(******************************************************************************************************************************************)
(****************************				             	Init / Reset Part                                                   *****************************)
(******************************************************************************************************************************************)
IF xSetEnd THEN
	xEnd:=TRUE;
	xInitStep:=FALSE;
	xSetEnd:=FALSE;
	xStop:=FALSE;
	xStartMainPrc:=FALSE;
	xInitMainCtr:=FALSE;
	xStartMainCtr:=FALSE;
	xStart:=FALSE;
	xHardwareError:=FALSE;
	xQuitErr:=FALSE;
	xError:=FALSE;
	iErrorNr:=0;
	xInitError:=FALSE;
	xFreeze:=FALSE;
	xAbord:=FALSE;
	xReset:=FALSE;
END_IF;
END_FUNCTION_BLOCK

(* POU PRG_STATION_LAYER3/FB_STATIONEN/FB_FUNCTION/FB_FctToolFeedReference, ST *)
FUNCTION_BLOCK FB_FctToolFeedReference
VAR_INPUT
	xMicroRodActive: BOOL;		(* choice of the machine MicroWire or MicroRod *)
	xBeckhoffDriveActive: BOOL;	(* choice of the axis Beckhoff or EcoStep *)
	xSafetyCircuitOn:BOOL;			(* state of the safety circuit-->TRUE=Machine current ON, FALSE=Machine current OFF *)
	T_Standard:ST_RETAIN_DATA;							(* Novram data structure for the standard process parameter *)
END_VAR
VAR_IN_OUT
	xStart : BOOL;					(* start the function *)
	xReset : BOOL;				(* reset the function *)
	xStop : BOOL;					(* stop the active function *)
	xQuitErr : BOOL;				(* quit the error caused of the active function *)
	xAbord : BOOL;				(* abord the active function *)
	TAxisToolFeeder:ST_AXIS;		(* data structure for the ToolFeeder axis *)
END_VAR
VAR_OUTPUT
	xEnd : BOOL;					(* state of the function if a active function is ended *)
	xError : BOOL;					(* state of the function if a active function caused an error *)
	iErrorNr : INT;					(* state of the function if a active function caused an error, in this case give the error number *)
END_VAR
VAR
	xHardwareError: BOOL := FALSE;
	xInitError: BOOL := FALSE;
	iStepError: INT := 0;
	xStartMainCtr: BOOL := FALSE;
	xStartMainPrc: BOOL := FALSE;
	xInitMainCtr: BOOL := FALSE;
	iStepPrc: INT := 0;
	xSetEnd: BOOL := FALSE;
	xInitStep: BOOL := FALSE;
	xFreeze: BOOL := FALSE;
	iTmpErrorNr:INT:=0;
	xTmpInit:BOOL;
	iTmp:INT;
END_VAR
(****************************************************************************************************************************************************)
(*******                                This Functionblock define the function for reference the ToolFeeder Axis                                                 ********)
(****************************************************************************************************************************************************)

(******************************************************************************************************************************************)
(****************************				           Reset Function Part                                                 *****************************)
(******************************************************************************************************************************************)
IF xReset AND NOT(xSetEnd) THEN
	xEnd:=FALSE;
	xSetEnd:=TRUE;
END_IF;
(******************************************************************************************************************************************)
(****************************				              Error Controlling Part                                            *****************************)
(******************************************************************************************************************************************)
IF (xHardwareError OR ((TAxisToolFeeder.T_CtrleSingle.xErr) AND xStartMainPrc)) AND NOT(xSetEnd) THEN
	IF NOT(TAxisToolFeeder.T_CtrleSingle.xExecute) THEN
		IF NOT(xInitError) THEN
			iStepError:=100;
			xInitError:=TRUE;
			IF xHardwareError THEN
				iErrorNr:=iTmpErrorNr;
			ELSE
				xHardwareError:=TRUE;	(* Hardware Error *)
			END_IF;
		END_IF;
		CASE iStepError OF
			100:	iStepError:=0;
				xError:=TRUE;
		END_CASE;
		IF xQuitErr THEN
			xSetEnd:=TRUE;
		END_IF;
	END_IF;
END_IF;
(******************************************************************************************************************************************)
(****************************				              Main Controlling Part                                            *****************************)
(******************************************************************************************************************************************)
IF (xStart OR xStartMainCtr) AND NOT(xSetEnd) AND NOT(xHardwareError) THEN
	IF NOT (xInitMainCtr) THEN
		iTmpErrorNr:=0;
		iStepPrc:=100;
		xInitMainCtr:=TRUE;
		xStartMainCtr:=TRUE;
		xStart:=FALSE;
		xEnd:=FALSE;
		xAbord:=FALSE;
		xTmpInit:=FALSE;
	END_IF;
	IF xStop AND NOT(xTmpInit) THEN
		xTmpInit:=TRUE;
		iTmp:=100;
		RETURN;
	END_IF;
	IF xFreeze THEN
		IF xStart AND NOT(xAbord) THEN
			xFreeze:=FALSE;
			xStart:=FALSE;
		END_IF;
		IF xAbord THEN
			xAbord:=FALSE;
			xFreeze:=FALSE;
			xStart:=FALSE;
			xSetEnd:=TRUE;
		END_IF;
		RETURN;
	END_IF;
	IF NOT(xStartMainPrc) AND NOT(xSetEnd) THEN
		xStartMainPrc:=TRUE;
	END_IF;
END_IF;
(******************************************************************************************************************************************)
(****************************				             immediate Stop Part                                              *****************************)
(******************************************************************************************************************************************)
IF xTmpInit AND NOT(xSetEnd) THEN
	IF NOT(xSafetyCircuitOn) THEN
		xTmpInit:=FALSE;
		iTmp:=100;
		xSetEnd:=TRUE;
		RETURN;
	END_IF;
	CASE iTmp OF
		100:	TAxisToolFeeder.T_CtrleSingle.iFunction:=5;
			TAxisToolFeeder.T_CtrleSingle.xExecute:=NOT(TAxisToolFeeder.T_CtrleSingle.xNotMoving);
			iTmp:=200;
			RETURN;
		200:	IF NOT(TAxisToolFeeder.T_CtrleSingle.xExecute) AND TAxisToolFeeder.T_CtrleSingle.xDone THEN
				iTmp:=300;
			END_IF;
			RETURN;
		300:	xTmpInit:=FALSE;
			iTmp:=100;
			xSetEnd:=TRUE;
			RETURN;
	END_CASE;
END_IF;
(******************************************************************************************************************************************)
(****************************				             Main Procedure Part                                             *****************************)
(******************************************************************************************************************************************)
IF xStartMainPrc AND NOT(xSetEnd) AND NOT(xHardwareError) THEN
	CASE iStepPrc OF
		100:	IF NOT(xInitStep) THEN
				xInitStep:=TRUE;
				IF NOT(TAxisToolFeeder.T_CtrleSingle.xDone)THEN
					xHardwareError:=TRUE;
					iTmpErrorNr:=1;
					RETURN;
				END_IF;
				IF NOT(TAxisToolFeeder.T_CtrleSingle.xPower) THEN
					TAxisToolFeeder.T_CtrleSingle.iFunction:=3;
					TAxisToolFeeder.T_CtrleSingle.xExecute:=TRUE;
				END_IF;
			END_IF;
			IF NOT(TAxisToolFeeder.T_CtrleSingle.xExecute) AND TAxisToolFeeder.T_CtrleSingle.xDone THEN
				xStartMainPrc:=FALSE;
				xInitStep:=FALSE;
				iStepPrc:=200;
			END_IF;
		200:	IF NOT(xInitStep) THEN
				xInitStep:=TRUE;
				TAxisToolFeeder.T_CtrleSingle.lrHomingMethode:=5;
				TAxisToolFeeder.T_CtrleSingle.lrHomeSpeedSwitch:=T_Standard.T_TeachINToolFeeder.rRefSpeed;
				TAxisToolFeeder.T_CtrleSingle.lrHomeSpeedZero:=T_Standard.T_TeachINToolFeeder.rRefSpeed / 10.0;
				TAxisToolFeeder.T_CtrleSingle.lrHomeAcceleration:=T_Standard.T_TeachINToolFeeder.rAcceleration;
				TAxisToolFeeder.T_CtrleSingle.iFunction:=9;	(* Reference Axis *)
				TAxisToolFeeder.T_CtrleSingle.xExecute:=TRUE;
			END_IF;
			IF NOT(TAxisToolFeeder.T_CtrleSingle.xExecute) AND TAxisToolFeeder.T_CtrleSingle.xDone THEN
				xStartMainPrc:=FALSE;
				xInitStep:=FALSE;
				iStepPrc:=0;
				xSetEnd:=TRUE;
			END_IF;
	END_CASE;
END_IF;
(******************************************************************************************************************************************)
(****************************				           Parallel Procedure Part                                          *****************************)
(******************************************************************************************************************************************)

(******************************************************************************************************************************************)
(****************************				             	Init / Reset Part                                                   *****************************)
(******************************************************************************************************************************************)
IF xSetEnd THEN
	xEnd:=TRUE;
	xInitStep:=FALSE;
	xSetEnd:=FALSE;
	xStop:=FALSE;
	xStartMainPrc:=FALSE;
	xInitMainCtr:=FALSE;
	xStartMainCtr:=FALSE;
	xStart:=FALSE;
	xHardwareError:=FALSE;
	xQuitErr:=FALSE;
	xError:=FALSE;
	iErrorNr:=0;
	xInitError:=FALSE;
	xFreeze:=FALSE;
	xAbord:=FALSE;
	xReset:=FALSE;
END_IF;
END_FUNCTION_BLOCK

(* POU PRG_STATION_LAYER3/FB_STATIONEN/FB_FUNCTION/FB_FctStopAxisMovement, ST *)
FUNCTION_BLOCK FB_FctStopAxisMovement
VAR_INPUT
	xMicroRodActive: BOOL;		(* choice of the machine MicroWire or MicroRod *)
	xBeckhoffDriveActive: BOOL;	(* choice of the axis Beckhoff or EcoStep *)
	xSafetyCircuitOn:BOOL;			(* state of the safety circuit-->TRUE=Machine current ON, FALSE=Machine current OFF *)
	T_ProcessImageData:ST_RETAIN_DATA_PROCESSIMAGE;	(* Novram data structure for the process parameter *)
	T_Standard:ST_RETAIN_DATA;							(* Novram data structure for the standard process parameter *)
END_VAR
VAR_IN_OUT
	xStart : BOOL;					(* start the function *)
	xReset : BOOL;				(* reset the function *)
	xStop : BOOL;					(* stop the active function *)
	xQuitErr : BOOL;				(* quit the error caused of the active function *)
	xAbord : BOOL;				(* abord the active function *)
	TAxisToolLeft:ST_AXIS;		(* data structure for the ToolLeft axis *)
	TAxisToolCenter:ST_AXIS;		(* data structure for the ToolCenter axis *)
	TAxisToolRight:ST_AXIS;		(* data structure for the ToolRight axis *)
	TAxisToolFeeder:ST_AXIS;		(* data structure for the ToolFeeder axis *)
	TAxisGrindFeeder:ST_AXIS;	(* data structure for the GrindFeeder axis *)
END_VAR
VAR_OUTPUT
	xEnd : BOOL;					(* state of the function if a active function is ended *)
	xError : BOOL;					(* state of the function if a active function caused an error *)
	iErrorNr : INT;					(* state of the function if a active function caused an error, in this case give the error number *)
END_VAR
VAR
	xHardwareError: BOOL := FALSE;
	xInitError: BOOL := FALSE;
	iStepError: INT := 0;
	xStartMainCtr: BOOL := FALSE;
	xStartMainPrc: BOOL := FALSE;
	xInitMainCtr: BOOL := FALSE;
	iStepPrc: INT := 0;
	xSetEnd: BOOL := FALSE;
	xInitStep: BOOL := FALSE;
	xFreeze: BOOL := FALSE;
	iTmpErrorNr:INT:=0;
	xTmpInit:BOOL;
	iTmp:INT;
	xTmp: BOOL;
	xReadFirstTime: BOOL;
	xTmp1: BOOL;
	rToolRotationSpeed: REAL;
	FBToolCalcul:FB_TOOL_CALCUL;
	rToolFeedLength: REAL;
	rToolDiameter: REAL;
	rGrindFeedPlunge: REAL;
	ii: INT;
	iStartSection: INT;
	iEndSection: INT;
	rSpeedGrindFeed: REAL;
	rSpeedToolFeed: REAL;
	rTimeGrindPlunge: REAL;
	FBCalcGearFactor: FB_CALC_GEARFACTOR;
	lrToolFeederActualPosition: LREAL;
	iTmpStartSection: INT;
	FBCalcPlungeGrinding: FB_CALC_PLUNGE_GRINDING;
	xResetFB: BOOL;
	xGrindFeedMaster: BOOL;
	xCheckToolFeedPosition: BOOL;
	lrToolFeederPosition: LREAL;
	lrToolRightPosition: LREAL;
	lrSaveToolFeederPosition: LREAL;
	lrSaveToolRightPosition: LREAL;
	rPlungeCycleGrindFeedGeometry: REAL;
END_VAR
(****************************************************************************************************************************************************)
(***********                               This Functionblock check the movement of all axis and stopp all movement                              ************)
(****************************************************************************************************************************************************)

IF NOT(xReadFirstTime) THEN
	xReadFirstTime:=TRUE;
END_IF;
(******************************************************************************************************************************************)
(****************************				           Reset Function Part                                                 *****************************)
(******************************************************************************************************************************************)
IF xReset AND NOT(xSetEnd) THEN
	xEnd:=FALSE;
	xSetEnd:=TRUE;
END_IF;
(******************************************************************************************************************************************)
(****************************				              Error Controlling Part                                            *****************************)
(******************************************************************************************************************************************)
xTmp:=	TAxisToolLeft.T_CtrleSingle.xErr OR
		(TAxisToolCenter.T_CtrleSingle.xErr AND xMicroRodActive) OR
		TAxisToolRight.T_CtrleSingle.xErr OR
		TAxisToolFeeder.T_CtrleSingle.xErr OR
		TAxisGrindFeeder.T_CtrleSingle.xErr;
xTmp1:=	NOT(TAxisToolLeft.T_CtrleSingle.xExecute) AND
		((NOT(TAxisToolCenter.T_CtrleSingle.xExecute) AND xMicroRodActive) OR NOT(xMicroRodActive)) AND
		 NOT(TAxisToolRight.T_CtrleSingle.xExecute) AND
		((NOT(TAxisToolFeeder.T_CtrleSingle.xExecute) AND NOT(xMicroRodActive)) OR xMicroRodActive) AND
		NOT(TAxisGrindFeeder.T_CtrleSingle.xExecute);
IF (xHardwareError OR (xTmp AND xStartMainPrc)) AND NOT(xSetEnd) THEN
	IF xTmp1 THEN
		IF NOT(xInitError) THEN
			iStepError:=100;
			xInitError:=TRUE;
			IF xHardwareError THEN
				iErrorNr:=iTmpErrorNr;
			ELSE
				xHardwareError:=TRUE;	(* Hardware Error *)
			END_IF;
		END_IF;
		CASE iStepError OF
			100:	iStepError:=0;
				xError:=TRUE;
		END_CASE;
		IF xQuitErr THEN
			xSetEnd:=TRUE;
		END_IF;
	END_IF;
END_IF;
(******************************************************************************************************************************************)
(****************************				              Main Controlling Part                                            *****************************)
(******************************************************************************************************************************************)
IF (xStart OR xStartMainCtr) AND NOT(xSetEnd) AND NOT(xHardwareError) THEN
	IF NOT (xInitMainCtr) THEN
		iTmpErrorNr:=0;
		iStepPrc:=100;
		xInitMainCtr:=TRUE;
		xStartMainCtr:=TRUE;
		xStart:=FALSE;
		xEnd:=FALSE;
		xAbord:=FALSE;
		xTmpInit:=FALSE;
		xCheckToolFeedPosition:=FALSE;
	END_IF;
	IF xStop AND NOT(xTmpInit) THEN
		xTmpInit:=TRUE;
		iTmp:=100;
		RETURN;
	END_IF;
	IF xFreeze THEN
		IF xStart AND NOT(xAbord) THEN
			xFreeze:=FALSE;
			xStart:=FALSE;
		END_IF;
		IF xAbord THEN
			xAbord:=FALSE;
			xFreeze:=FALSE;
			xStart:=FALSE;
			xSetEnd:=TRUE;
		END_IF;
		RETURN;
	END_IF;
	IF NOT(xStartMainPrc) AND NOT(xSetEnd) THEN
		xStartMainPrc:=TRUE;
	END_IF;
END_IF;
(******************************************************************************************************************************************)
(****************************				             immediate Stop Part                                              *****************************)
(******************************************************************************************************************************************)
IF xTmpInit AND NOT(xSetEnd) THEN
	IF NOT(xSafetyCircuitOn) THEN
		xTmpInit:=FALSE;
		iTmp:=100;
		xSetEnd:=TRUE;
		RETURN;
	END_IF;
	CASE iTmp OF
		100:	TAxisToolLeft.T_CtrleSingle.iFunction:=5;
			TAxisToolLeft.T_CtrleSingle.xExecute:=NOT(TAxisToolLeft.T_CtrleSingle.xNotMoving);
			IF xMicroRodActive THEN
				TAxisToolCenter.T_CtrleSingle.iFunction:=5;
				TAxisToolCenter.T_CtrleSingle.xExecute:=NOT(TAxisToolCenter.T_CtrleSingle.xNotMoving);
			END_IF;
			TAxisToolRight.T_CtrleSingle.iFunction:=5;
			TAxisToolRight.T_CtrleSingle.xExecute:=NOT(TAxisToolRight.T_CtrleSingle.xNotMoving);
			TAxisToolFeeder.T_CtrleSingle.iFunction:=5;
			TAxisToolFeeder.T_CtrleSingle.xExecute:=NOT(TAxisToolFeeder.T_CtrleSingle.xNotMoving);
			TAxisGrindFeeder.T_CtrleSingle.iFunction:=5;
			TAxisGrindFeeder.T_CtrleSingle.xExecute:=NOT(TAxisGrindFeeder.T_CtrleSingle.xNotMoving);
			iTmp:=200;
			RETURN;
		200:	xTmp:=	NOT(TAxisToolLeft.T_CtrleSingle.xExecute) AND TAxisToolLeft.T_CtrleSingle.xDone AND
					((NOT(TAxisToolCenter.T_CtrleSingle.xExecute) AND TAxisToolCenter.T_CtrleSingle.xDone AND xMicroRodActive) OR NOT(xMicroRodActive)) AND
					NOT(TAxisToolRight.T_CtrleSingle.xExecute) AND TAxisToolRight.T_CtrleSingle.xDone AND
					NOT(TAxisToolFeeder.T_CtrleSingle.xExecute) AND TAxisToolFeeder.T_CtrleSingle.xDone AND
					NOT(TAxisGrindFeeder.T_CtrleSingle.xExecute) AND TAxisGrindFeeder.T_CtrleSingle.xDone;
			IF xTmp THEN
				iTmp:=300;
			END_IF;
			RETURN;
		300:	IF xMicroRodActive THEN
				IF TAxisToolCenter.T_CtrleSingle.xSlave THEN
					TAxisToolCenter.T_CtrleSingle.iFunction:=25;
					TAxisToolCenter.T_CtrleSingle.xExecute:=TRUE;
				END_IF;
			END_IF;
			IF TAxisToolRight.T_CtrleSingle.xSlave THEN
				TAxisToolRight.T_CtrleSingle.iFunction:=25;
				TAxisToolRight.T_CtrleSingle.xExecute:=TRUE;
			END_IF;
			IF TAxisToolFeeder.T_CtrleSingle.xSlave THEN
				TAxisToolFeeder.T_CtrleSingle.iFunction:=25;
				TAxisToolFeeder.T_CtrleSingle.xExecute:=TRUE;
			END_IF;
			IF TAxisGrindFeeder.T_CtrleSingle.xSlave THEN
				TAxisGrindFeeder.T_CtrleSingle.iFunction:=25;
				TAxisGrindFeeder.T_CtrleSingle.xExecute:=TRUE;
			END_IF;
			iTmp:=400;
			RETURN;
		400:	xTmp:=	((NOT(TAxisToolCenter.T_CtrleSingle.xExecute) AND TAxisToolCenter.T_CtrleSingle.xDone AND xMicroRodActive) OR NOT(xMicroRodActive)) AND
					NOT(TAxisToolRight.T_CtrleSingle.xExecute) AND TAxisToolRight.T_CtrleSingle.xDone AND
					NOT(TAxisToolFeeder.T_CtrleSingle.xExecute) AND TAxisToolFeeder.T_CtrleSingle.xDone AND
					NOT(TAxisGrindFeeder.T_CtrleSingle.xExecute) AND TAxisGrindFeeder.T_CtrleSingle.xDone;
			IF xTmp THEN
				iTmp:=500;
			END_IF;
			RETURN;
		500:	xTmpInit:=FALSE;
			iTmp:=100;
			xSetEnd:=TRUE;
			RETURN;
	END_CASE;
END_IF;
(******************************************************************************************************************************************)
(****************************				             Main Procedure Part                                             *****************************)
(******************************************************************************************************************************************)
IF xStartMainPrc AND NOT(xSetEnd) AND NOT(xHardwareError) THEN
	CASE iStepPrc OF
		(* Initial Procedure *)
		100:	IF NOT(xInitStep) THEN
				xInitStep:=TRUE;
				TAxisToolLeft.T_CtrleSingle.iFunction:=5;
				TAxisToolLeft.T_CtrleSingle.xExecute:=NOT(TAxisToolLeft.T_CtrleSingle.xNotMoving);
				IF xMicroRodActive THEN
					TAxisToolCenter.T_CtrleSingle.iFunction:=5;
					TAxisToolCenter.T_CtrleSingle.xExecute:=NOT(TAxisToolCenter.T_CtrleSingle.xNotMoving);
				END_IF;
				TAxisToolRight.T_CtrleSingle.iFunction:=5;
				TAxisToolRight.T_CtrleSingle.xExecute:=NOT(TAxisToolRight.T_CtrleSingle.xNotMoving);
				TAxisToolFeeder.T_CtrleSingle.iFunction:=5;
				TAxisToolFeeder.T_CtrleSingle.xExecute:=NOT(TAxisToolFeeder.T_CtrleSingle.xNotMoving);
				TAxisGrindFeeder.T_CtrleSingle.iFunction:=5;
				TAxisGrindFeeder.T_CtrleSingle.xExecute:=NOT(TAxisGrindFeeder.T_CtrleSingle.xNotMoving);
			END_IF;
			xTmp:=	NOT(TAxisToolLeft.T_CtrleSingle.xExecute) AND TAxisToolLeft.T_CtrleSingle.xDone AND
					((NOT(TAxisToolCenter.T_CtrleSingle.xExecute) AND TAxisToolCenter.T_CtrleSingle.xDone AND xMicroRodActive) OR NOT(xMicroRodActive)) AND
					NOT(TAxisToolRight.T_CtrleSingle.xExecute) AND TAxisToolRight.T_CtrleSingle.xDone AND
					NOT(TAxisToolFeeder.T_CtrleSingle.xExecute) AND TAxisToolFeeder.T_CtrleSingle.xDone AND
					NOT(TAxisGrindFeeder.T_CtrleSingle.xExecute) AND TAxisGrindFeeder.T_CtrleSingle.xDone;
			IF xTmp THEN
				xStartMainPrc:=FALSE;
				xInitStep:=FALSE;
				iStepPrc:=200;
			END_IF;
		200:	IF NOT(xInitStep) THEN
				xInitStep:=TRUE;
				IF xMicroRodActive THEN
					IF TAxisToolCenter.T_CtrleSingle.xSlave THEN
						TAxisToolCenter.T_CtrleSingle.iFunction:=25;
						TAxisToolCenter.T_CtrleSingle.xExecute:=TRUE;
					END_IF;
				END_IF;
				IF TAxisToolRight.T_CtrleSingle.xSlave THEN
					TAxisToolRight.T_CtrleSingle.iFunction:=25;
					TAxisToolRight.T_CtrleSingle.xExecute:=TRUE;
				END_IF;
				IF TAxisToolFeeder.T_CtrleSingle.xSlave THEN
					TAxisToolFeeder.T_CtrleSingle.iFunction:=25;
					TAxisToolFeeder.T_CtrleSingle.xExecute:=TRUE;
				END_IF;
				IF TAxisGrindFeeder.T_CtrleSingle.xSlave THEN
					TAxisGrindFeeder.T_CtrleSingle.iFunction:=25;
					TAxisGrindFeeder.T_CtrleSingle.xExecute:=TRUE;
				END_IF;
			END_IF;
			xTmp:=	((NOT(TAxisToolCenter.T_CtrleSingle.xExecute) AND TAxisToolCenter.T_CtrleSingle.xDone AND xMicroRodActive) OR NOT(xMicroRodActive)) AND
					NOT(TAxisToolRight.T_CtrleSingle.xExecute) AND TAxisToolRight.T_CtrleSingle.xDone AND
					NOT(TAxisToolFeeder.T_CtrleSingle.xExecute) AND TAxisToolFeeder.T_CtrleSingle.xDone AND
					NOT(TAxisGrindFeeder.T_CtrleSingle.xExecute) AND TAxisGrindFeeder.T_CtrleSingle.xDone;
			IF xTmp THEN
				(* Procedure is finished *)
				xStartMainPrc:=FALSE;
				xInitStep:=FALSE;
				iStepPrc:=0;
				xSetEnd:=TRUE;
			END_IF;
	END_CASE;
END_IF;
(******************************************************************************************************************************************)
(****************************				           Parallel Procedure Part                                          *****************************)
(******************************************************************************************************************************************)
(******************************************************************************************************************************************)
(****************************				             	Init / Reset Part                                                   *****************************)
(******************************************************************************************************************************************)
IF xSetEnd THEN
	xEnd:=TRUE;
	xInitStep:=FALSE;
	xSetEnd:=FALSE;
	xStop:=FALSE;
	xStartMainPrc:=FALSE;
	xInitMainCtr:=FALSE;
	xStartMainCtr:=FALSE;
	xStart:=FALSE;
	xHardwareError:=FALSE;
	xQuitErr:=FALSE;
	xError:=FALSE;
	iErrorNr:=0;
	xInitError:=FALSE;
	xFreeze:=FALSE;
	xAbord:=FALSE;
	xReset:=FALSE;
	xCheckToolFeedPosition:=FALSE;
END_IF;
END_FUNCTION_BLOCK

(* POU PRG_HARDWARE_LAYER2/PRG_HW_GENERAL, FBD *)
PROGRAM PRG_HW_GENERAL
VAR
	FBHWHdd: FBHW_HDD;
	FBNovRam: FBHW_NOVRAM;
	FBDeviceId:FBHW_DEVICEID;
	FBBoxId:FBHW_BOXID;
	FBProfileFile: FB_PROFILE_FILE;
	FBControlLamp: FB_CONTROLLAMP;
	xDeleteThisVariable:BOOL;
END_VAR
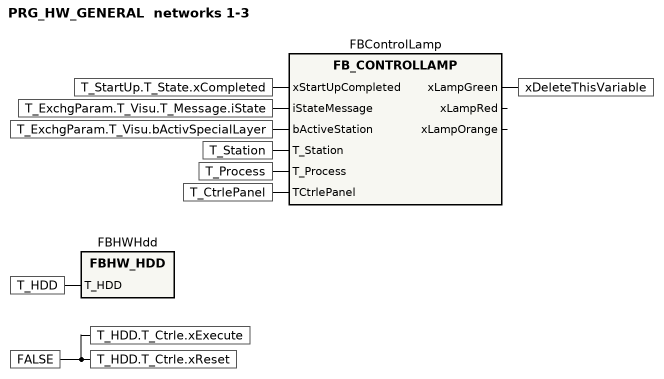
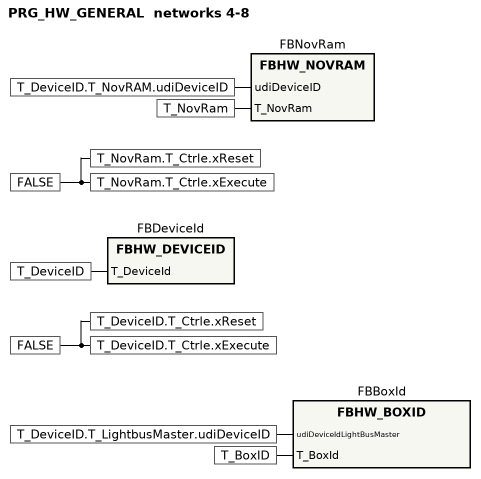
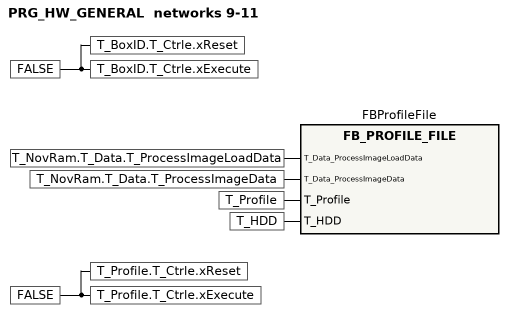
_FBD_ (* Function Block Diagram *)
NETWORK 1
	FBControlLamp:FB_CONTROLLAMP(xStartUpCompleted: T_StartUp.T_State.xCompleted, iStateMessage: T_ExchgParam.T_Visu.T_Message.iState, bActiveStation: T_ExchgParam.T_Visu.bActivSpecialLayer, T_Station: T_Station, T_Process: T_Process, TCtrlePanel: T_CtrlePanel) => xDeleteThisVariable
NETWORK 2
	FBHWHdd:FBHW_HDD(T_HDD: T_HDD)
NETWORK 3
	FALSE => T_HDD.T_Ctrle.xExecute, T_HDD.T_Ctrle.xReset
NETWORK 4
	FBNovRam:FBHW_NOVRAM(udiDeviceID: T_DeviceID.T_NovRAM.udiDeviceID, T_NovRam: T_NovRam)
NETWORK 5
	FALSE => T_NovRam.T_Ctrle.xReset, T_NovRam.T_Ctrle.xExecute
NETWORK 6
	FBDeviceId:FBHW_DEVICEID(T_DeviceId: T_DeviceID)
NETWORK 7
	FALSE => T_DeviceID.T_Ctrle.xReset, T_DeviceID.T_Ctrle.xExecute
NETWORK 8
	FBBoxId:FBHW_BOXID(udiDeviceIdLightBusMaster: T_DeviceID.T_LightbusMaster.udiDeviceID, T_BoxId: T_BoxID)
NETWORK 9
	FALSE => T_BoxID.T_Ctrle.xReset, T_BoxID.T_Ctrle.xExecute
NETWORK 10
	FBProfileFile:FB_PROFILE_FILE(T_Data_ProcessImageLoadData: T_NovRam.T_Data.T_ProcessImageLoadData, T_Data_ProcessImageData: T_NovRam.T_Data.T_ProcessImageData, T_Profile: T_Profile, T_HDD: T_HDD)
NETWORK 11
	FALSE => T_Profile.T_Ctrle.xReset, T_Profile.T_Ctrle.xExecute
_END_FBD_
(* the same logic as Structured Text *)
(* Network 1 *)
FBControlLamp(xStartUpCompleted := T_StartUp.T_State.xCompleted, iStateMessage := T_ExchgParam.T_Visu.T_Message.iState, bActiveStation := T_ExchgParam.T_Visu.bActivSpecialLayer, T_Station := T_Station, T_Process := T_Process, TCtrlePanel := T_CtrlePanel);
xDeleteThisVariable := FBControlLamp.xLampGreen;
(* Network 2 *)
FBHWHdd(T_HDD := T_HDD);
(* Network 3 *)
T_HDD.T_Ctrle.xExecute := FALSE;
T_HDD.T_Ctrle.xReset := FALSE;
(* Network 4 *)
FBNovRam(udiDeviceID := T_DeviceID.T_NovRAM.udiDeviceID, T_NovRam := T_NovRam);
(* Network 5 *)
T_NovRam.T_Ctrle.xReset := FALSE;
T_NovRam.T_Ctrle.xExecute := FALSE;
(* Network 6 *)
FBDeviceId(T_DeviceId := T_DeviceID);
(* Network 7 *)
T_DeviceID.T_Ctrle.xReset := FALSE;
T_DeviceID.T_Ctrle.xExecute := FALSE;
(* Network 8 *)
FBBoxId(udiDeviceIdLightBusMaster := T_DeviceID.T_LightbusMaster.udiDeviceID, T_BoxId := T_BoxID);
(* Network 9 *)
T_BoxID.T_Ctrle.xReset := FALSE;
T_BoxID.T_Ctrle.xExecute := FALSE;
(* Network 10 *)
FBProfileFile(T_Data_ProcessImageLoadData := T_NovRam.T_Data.T_ProcessImageLoadData, T_Data_ProcessImageData := T_NovRam.T_Data.T_ProcessImageData, T_Profile := T_Profile, T_HDD := T_HDD);
(* Network 11 *)
T_Profile.T_Ctrle.xReset := FALSE;
T_Profile.T_Ctrle.xExecute := FALSE;
END_PROGRAM

(* POU FB_HARDWARE/FBHW_HDD, ST *)
FUNCTION_BLOCK FBHW_HDD
VAR_INPUT
END_VAR
VAR_OUTPUT
END_VAR
VAR_IN_OUT
	T_HDD:ST_HDD;
END_VAR
VAR
(* variable *)
	xConfirmResetFB: BOOL;
	i:INT;
	dwOpenFileMod:DWORD;
	udiHdleFile:UINT;
	xFileOpen: BOOL;
	xFileClose:BOOL;
	xFileRead:BOOL;
	xFileAppendWrite:BOOL;
	xFileCreate:BOOL;
	xFileBiggerAsMaxLine:BOOL;
	xFileDelete: BOOL;
	xRenameFile:BOOL;

(* function bloc *)
	fbFileOpen:FB_FileOpen;
	fbFileWrite:FB_FileWrite;

	fbFileClose:FB_FileClose;
	fbFileGets:FB_FileGets;
	fbFilePuts:FB_FilePuts;

	fbFileDelete:FB_FileDelete;
	fbRenameFile:FB_FileRename;
(* Trigger *)
	RisingEdgeExecute:R_TRIG;
	RisingEdgeReset:R_TRIG;
END_VAR
(****************************************************************************************************************************************************)
(***********                                                  This Functionblock is for manage the file handling                                                             ************)
(****************************************************************************************************************************************************)
(* waiting for reset *)
	RisingEdgeReset(CLK:=T_HDD.T_Ctrle.xReset);
	IF RisingEdgeReset.Q THEN
	(* init. function bloc *)
		fbFileOpen(bExecute:=FALSE);
		fbFileClose(bExecute:=FALSE);
		fbFileWrite(bExecute:=FALSE);
		fbFileGets(bExecute:=FALSE);
		fbFilePuts(bExecute:=FALSE);
		fbFileDelete(bExecute:=FALSE);
		fbRenameFile(bExecute:=FALSE);
	(* init. variable *)
		dwOpenFileMod:=0;
		udiHdleFile:=0;
		xFileOpen:=FALSE;
		xFileClose:=FALSE;
		xFileRead:=FALSE;
		xFileAppendWrite:=FALSE;
		xFileCreate:=FALSE;
		xFileBiggerAsMaxLine:=FALSE;
		xFileDelete:=FALSE;
		xRenameFile:=FALSE;
	(* init. structure *)
		T_HDD.T_Ctrle.xDone:=FALSE;
		T_HDD.T_Ctrle.xErr:=FALSE;
		T_HDD.T_Ctrle.udiErrorID:=0;
		T_HDD.T_Ctrle.iFunction:=0;
		T_HDD.T_File.sPathAndFileName:='';
		T_HDD.T_File.sOldPathAndFileName:='';
		T_HDD.T_Ctrle.tTimeOut:=T#2s;
		T_HDD.T_Ctrle.xLocked:=FALSE;
		(* set flag done *)
		xConfirmResetFB:=TRUE;
		(* exit function *)
		RETURN;
	ELSE
		IF xConfirmResetFB THEN
		(* confirm reset FB *)
			T_HDD.T_Ctrle.xDone:=TRUE;
			T_HDD.T_Ctrle.xErr:=FALSE;
			T_HDD.T_Ctrle.udiErrorID:=0;
			T_HDD.T_Ctrle.xLocked:=FALSE;
			(* init. variable *)
			xConfirmResetFB:=FALSE;
		END_IF
	END_IF

(* waiting for execute *)
	RisingEdgeExecute(CLK:=T_HDD.T_Ctrle.xExecute);
	IF RisingEdgeExecute.Q THEN
		CASE T_HDD.T_Ctrle.iFunction OF
		(* Read file *)
		1:	(* activ file open *)
			xFileOpen:=TRUE;
			dwOpenFileMod:=FOPEN_MODEREAD OR FOPEN_MODEPLUS OR FOPEN_MODETEXT;
		(* Write file *)
		2:	(* activ file open *)
			xFileOpen:=TRUE;
			dwOpenFileMod:=FOPEN_MODEWRITE OR FOPEN_MODEPLUS OR FOPEN_MODETEXT;
		(* overwrite file *)
		3:	(* activ file open *)
			xFileOpen:=TRUE;
			dwOpenFileMod:=FOPEN_MODEAPPEND OR FOPEN_MODEPLUS OR FOPEN_MODETEXT;
		(* file exists *)
		4:	(* activ file open *)
			xFileOpen:=TRUE;
			dwOpenFileMod:=FOPEN_MODEREAD OR FOPEN_MODEPLUS OR FOPEN_MODETEXT;
		(* delete file *)
		5:	xFileDelete:=TRUE;
		(* rename file *)
		6:	xRenameFile:=TRUE;
		ELSE
		(* function not implemented *)
			 T_HDD.T_Ctrle.xDone:=FALSE;
			 T_HDD.T_Ctrle.xErr:=TRUE;
			 T_HDD.T_Ctrle.udiErrorID:=16#F000;
			 T_HDD.T_Ctrle.xLocked:=FALSE;
			 (* exit FB *)
			 RETURN;
		END_CASE
		(* Init. variable *)
		T_HDD.T_Ctrle.xDone:=FALSE;
		T_HDD.T_Ctrle.xErr:=FALSE;
		T_HDD.T_Ctrle.udiErrorID:=16#0;
		xFileBiggerAsMaxLine:=FALSE;
		(* init. variable*)
		i:=1;
		RETURN;
	END_IF

(* Open file *)
	IF xFileOpen THEN
		fbFileOpen(	sNetId:=T_HDD.T_Config.sNetId,
					sPathName:=T_HDD.T_File.sPathAndFileName,
					nMode:=dwOpenFileMod,
					bExecute:=TRUE,
					tTimeout:=T#2s);
		IF NOT(fbFileOpen.bBusy) OR fbFileOpen.bError THEN
			IF NOT(fbFileOpen.bError) THEN
				CASE T_HDD.T_Ctrle.iFunction OF
				1:	xFileRead:=TRUE;
				2:	xFileCreate:=TRUE;
				3: 	xFileAppendWrite:=TRUE;
				4:	xFileClose:=TRUE;
				END_CASE
				(* Handle file *)
				udiHdleFile:=fbFileOpen.hFile;
			ELSE
				udiHdleFile:=0;
				 T_HDD.T_Ctrle.xDone:= FALSE;
				 T_HDD.T_Ctrle.xErr:=fbFileOpen.bError;
				 T_HDD.T_Ctrle.udiErrorID:=fbFileOpen.nErrId;
				 T_HDD.T_Ctrle.xLocked:=FALSE;
			END_IF
			(* set flag xfileopen off *)
			xFileOpen:=FALSE;
		END_IF
	ELSE fbFileOpen(bExecute:=FALSE); END_IF

(* Read file *)
	IF xFileRead THEN
		fbFileGets(	sNetId:=T_HDD.T_Config.sNetId,
					hFile:=udiHdleFile,
					bExecute:=TRUE,
					tTimeOut:=T_HDD.T_Ctrle.tTimeOut);
		IF NOT(fbFileGets.bBusy) OR fbFileGets.bError THEN
			T_HDD.T_Data.sData[i]:=fbFileGets.sLine;
			(* check eof or error *)
			IF fbFileGets.bEOF OR fbFileGets.bError OR i = csiMaxFileLine THEN
				 (* set flag xFileRead off *)
				 xFileRead:=FALSE;
				 (* activ closing file *)
				 xFileClose:=TRUE;
				 (* activ variable file bigger as structure *)
				 IF i = csiMaxFileLine THEN xFileBiggerAsMaxLine:=TRUE; END_IF
			ELSE
			(* read next line *)
				fbFileGets(bExecute:=FALSE);
				i:=i+1;
			END_IF
		END_IF
	ELSE fbFileGets(bExecute:=FALSE); END_IF

(* Write at the end of file or create file *)
	IF xFileAppendWrite OR xFileCreate THEN
		fbFilePuts(	sNetId:=T_HDD.T_Config.sNetId,
					hFile:=udiHdleFile,
					sLine:=CONCAT(T_HDD.T_Data.sData[i],'$L'),
					bExecute:=TRUE,
					tTimeOut:=T_HDD.T_Ctrle.tTimeOut);
		IF NOT(fbFilePuts.bBusy) OR fbFilePuts.bError THEN
			IF T_HDD.T_Data.sData[i+1] = '' THEN
				 (* set flag xFileCreate or xFileAppendWrite off *)
				xFileAppendWrite:=FALSE;
				xFileCreate:=FALSE;
				 (* activ closing file *)
				 xFileClose:=TRUE;
			ELSE
			(* Init. FB *)
				 fbFilePuts(bExecute:=FALSE);
				 (* next line *)
				i:=i+1;
			END_IF
		END_IF
	ELSE IF NOT(xFileAppendWrite) AND NOT(xFileCreate) THEN fbFilePuts(bExecute:=FALSE); END_IF
	END_IF

(* Close file *)
	IF xFileClose THEN
		fbFileClose(	sNetId:=T_HDD.T_Config.sNetId,
					hFile:=udiHdleFile,
					bExecute:=TRUE,
					tTimeout:=T#2s);
		IF NOT(fbFileClose.bBusy) OR fbFileClose.bError THEN
			 T_HDD.T_Ctrle.xDone:= NOT(fbFileClose.bBusy);
			 T_HDD.T_Ctrle.xErr:=fbFileClose.bError;
			 T_HDD.T_Ctrle.udiErrorID:=fbFileClose.nErrId;
			T_HDD.T_Ctrle.xLocked:=FALSE;
			 udiHdleFile:=0;
			(* check if file bigger as maximum reading line *)
			IF xFileBiggerAsMaxLine THEN
				T_HDD.T_Ctrle.xErr:=TRUE;
				T_HDD.T_Ctrle.udiErrorID:=16#F501;
			END_IF
			 (* set flag xFileClose off *)
			 xFileClose:=FALSE;
		END_IF
	ELSE fbFileClose(bExecute:=FALSE); END_IF

(* Delete file *)
	IF xFileDelete THEN
		fbFileDelete(	sNetId:=T_HDD.T_Config.sNetId,
					sPathName:=T_HDD.T_File.sPathAndFileName,
					bExecute:=TRUE,
					tTimeout:=T#2s);
		IF NOT(fbFileDelete.bBusy) OR fbFileDelete.bError THEN
			 T_HDD.T_Ctrle.xDone:= NOT(fbFileDelete.bBusy);
			 T_HDD.T_Ctrle.xErr:=fbFileDelete.bError;
			 T_HDD.T_Ctrle.udiErrorID:=fbFileDelete.nErrId;
			T_HDD.T_Ctrle.xLocked:=FALSE;
			 (* set flag xFileDelete off *)
			 xFileDelete:=FALSE;
		END_IF
	ELSE fbFileDelete(bExecute:=FALSE); END_IF

(* rename file *)
	IF xRenameFile THEN
		fbRenameFile(	sNetId:=T_HDD.T_Config.sNetId,
						sOldName:=T_HDD.T_File.sOldPathAndFileName,
						sNewName:=T_HDD.T_File.sPathAndFileName,
						ePath:=PATH_GENERIC,
						bExecute:=TRUE,
						tTimeout:=T#2s);
		IF NOT(fbRenameFile.bBusy) OR fbRenameFile.bError THEN
			 T_HDD.T_Ctrle.xDone:= NOT(fbRenameFile.bBusy);
			 T_HDD.T_Ctrle.xErr:=fbRenameFile.bError;
			 T_HDD.T_Ctrle.udiErrorID:=fbRenameFile.nErrId;
			T_HDD.T_Ctrle.xLocked:=FALSE;
			 (* set flag xFileDelete off *)
			 xRenameFile:=FALSE;
		END_IF
	ELSE fbRenameFile(bExecute:=FALSE); END_IF
END_FUNCTION_BLOCK

(* POU FB_HARDWARE/FBHW_NOVRAM, ST *)
FUNCTION_BLOCK FBHW_NOVRAM
VAR_INPUT
	udiDeviceID:UDINT;
END_VAR
VAR_IN_OUT
	T_NovRam:ST_NOVRAM;
END_VAR
VAR_OUTPUT
END_VAR
VAR
(* function bloc *)
	fbNovRamReadWrite:FB_NovRamReadWrite;
(* trigger *)
	RisingEdgeResetFB:R_TRIG;
	RisingEdgeExecute:R_TRIG;
(* variable *)
	xRead:BOOL:=FALSE;
	xWrite:BOOL:=FALSE;
	xConfirmResetFB: BOOL;
	xDummy1: BOOL;
	xDummy2: BOOL;
END_VAR
(****************************************************************************************************************************************************)
(***********                                            This Functionblock is for manage the NovRAM handling                                                      ************)
(****************************************************************************************************************************************************)
(* reset *)
	RisingEdgeResetFB(CLK:=T_NovRam.T_Ctrle.xReset);
	IF RisingEdgeResetFB.Q THEN
	(* init. variable *)
		xRead:=FALSE;
		xWrite:=FALSE;
	(* activ confirmation reset *)
		xConfirmResetFB:=TRUE;
	(* Exit FB *)
		RETURN;
	ELSE
		IF xConfirmResetFB THEN
		(* confirm reset FB *)
			T_NovRam.T_Ctrle.xFirstRead:=FALSE;
			T_NovRam.T_Ctrle.xDone:=TRUE;
			T_NovRam.T_Ctrle.xErr:=FALSE;
			T_NovRam.T_Ctrle.udiErrorID:=16#0;
		(* reset variable *)
			xConfirmResetFB:=FALSE;
		END_IF
	END_IF

(* execute *)
	RisingEdgeExecute(CLK:=T_NovRam.T_Ctrle.xExecute);
	IF RisingEdgeExecute.Q THEN
		(* init. capacity and pointer *)
		T_NovRam.T_Ctrle.udipSrcAddr:=ADR(T_NovRam.T_Data);
		T_NovRam.T_Ctrle.udiSrcLen:=SIZEOF(T_NovRam.T_Data);
		T_NovRam.T_Ctrle.udipDestAddr:=ADR(T_NovRam.T_Data);
		T_NovRam.T_Ctrle.udiDestLen:=SIZEOF(T_NovRam.T_Data);
		CASE T_NovRam.T_Ctrle.iFunction OF
		(* Read *)
		1:	xRead:=TRUE;
		(* Write *)
		2:	xWrite:=TRUE;
		ELSE
		(* function not implemented *)
			T_NovRam.T_Ctrle.xDone:=FALSE;
			T_NovRam.T_Ctrle.xErr:=TRUE;
			T_NovRam.T_Ctrle.udiErrorID:=16#F000;
			(* Exit FB *)
			RETURN;
		END_CASE
		(* Init. variable *)
		T_NovRam.T_Ctrle.xDone:=FALSE;
		T_NovRam.T_Ctrle.xErr:=FALSE;
		T_NovRam.T_Ctrle.udiErrorID:=0;
	(* Exit FB *)
		RETURN;
	END_IF

(* wait for read/write *)
	IF xRead OR xWrite THEN
		IF xWrite THEN
			xDummy1:=TRUE;
			xDummy2:=FALSE;
		END_IF;
		IF xRead THEN
			xDummy2:=TRUE;
			xDummy1:=FALSE;
		END_IF;
		fbNovRamReadWrite(	nDevId:=udiDeviceID,
							bRead:=xRead,
							bWrite:=xWrite,
							cbSrcLen:=T_NovRam.T_Ctrle.udiSrcLen,
							cbDestLen:=T_NovRam.T_Ctrle.udiDestLen,
							pSrcAddr:=T_NovRam.T_Ctrle.udipSrcAddr,
							pDestAddr:=T_NovRam.T_Ctrle.udipDestAddr,
							tTimeOut:=T_NovRam.T_Ctrle.tTimeOut);
		IF NOT(fbNovRamReadWrite.bBusy) OR fbNovRamReadWrite.bError THEN
			IF fbNovRamReadWrite.bError THEN
			(* set error *)
				T_NovRam.T_Ctrle.xDone:=FALSE;
				T_NovRam.T_Ctrle.xErr:=TRUE;
				T_NovRam.T_Ctrle.udiErrorID:=fbNovRamReadWrite.nErrId;
			ELSE
			(* confirm execution *)
				IF xRead THEN
					IF NOT(T_NovRam.T_Ctrle.xBlockReadFirstTime) THEN
						T_NovRam.T_Ctrle.xFirstRead:=TRUE;
					ELSE
						T_NovRam.T_Ctrle.xFirstRead:=FALSE;
					END_IF;
					T_NovRam.T_Ctrle.xBlockReadFirstTime:=FALSE;
				END_IF
				T_NovRam.T_Ctrle.xDone:=TRUE;
				T_NovRam.T_Ctrle.xErr:=FALSE;
				T_NovRam.T_Ctrle.udiErrorID:=0;
			END_IF
			(* reset variable *)
			xRead:=FALSE;
			xWrite:=FALSE;
		END_IF
	ELSE
		fbNovRamReadWrite(	nDevId:=udiDeviceID,
							bRead:=FALSE,
							bWrite:=FALSE);
	END_IF
END_FUNCTION_BLOCK

(* POU FB_HARDWARE/FBHW_DEVICEID, ST *)
FUNCTION_BLOCK FBHW_DEVICEID
VAR_INPUT
END_VAR
VAR_IN_OUT
	T_DeviceId:ST_DEVICEID;
END_VAR
VAR_OUTPUT
END_VAR
VAR
(* pointer of Device ID *)
	ptrDeviceId: POINTER TO ST_DEVICEID;
(* function bloc *)
	FBGeviceInfoByName:IOF_GetDeviceInfoByName;
(* trigger *)
	RisingEdgeResetFB:R_TRIG;
	RisingEdgeExecute:R_TRIG;
	FallingEdgeBusy:F_TRIG;
(* variable *)
	xGetDeviceId:BOOL:=FALSE;
	xConfirmResetFB:BOOL:=FALSE;
	iPtrDeviceName:INT:=0;
	T_DeviceId_AdrTmp:ARRAY[1..10] OF ST_DEVICEID_DATA_ADR;
	xInitReadStructure: BOOL;
	xCopyReadyStructure:BOOL;
END_VAR
(****************************************************************************************************************************************************)
(***********                                                This Functionblock is for init the Beckhoff component                                                          ************)
(****************************************************************************************************************************************************)
(* reset *)
	RisingEdgeResetFB(CLK:=T_DeviceId.T_Ctrle.xReset);
	IF RisingEdgeResetFB.Q THEN
	(* init ptr*)
		ptrDeviceId:=ADR(T_DeviceId);
	(* init. variable *)
		xGetDeviceId:=FALSE;
		iPtrDeviceName:=1;
	(* Init. variable *)
		ptrDeviceId^.T_Ctrle.xDone:=FALSE;
		ptrDeviceId^.T_Ctrle.xErr:=FALSE;
		ptrDeviceId^.T_Ctrle.udiErrorID:=0;
	(* activ confirm reset *)
		xConfirmResetFB:=TRUE;
	(* Exit FB *)
		RETURN;
	ELSE
		IF xConfirmResetFB THEN
		(* confirm reset FB *)
			ptrDeviceId^.T_Ctrle.xDone:=TRUE;
			ptrDeviceId^.T_Ctrle.xErr:=FALSE;
			ptrDeviceId^.T_Ctrle.udiErrorID:=0;
		(* reset variable *)
			xConfirmResetFB:=FALSE;
		END_IF
	END_IF

(* execute *)
	RisingEdgeExecute(CLK:=T_DeviceId.T_Ctrle.xExecute);
	IF RisingEdgeExecute.Q THEN
	(* init ptr*)
		ptrDeviceId:=ADR(T_DeviceId);
		ptrDeviceId^.T_Ctrle.xDone:=FALSE;
		ptrDeviceId^.T_Ctrle.xErr:=FALSE;
		ptrDeviceId^.T_Ctrle.udiErrorID:=0;
	(* activ get device Id *)
		xInitReadStructure:=TRUE;
	(* Exit FB *)
		RETURN;
	END_IF

(* init. read structure *)
	IF xInitReadStructure THEN
	(* PLC name *)
		T_DeviceId_AdrTmp[1]:=T_DeviceId.T_CX1020;
		(* feldbus name *)
		T_DeviceId_AdrTmp[2]:=T_DeviceId.T_CANOpenMaster;
		T_DeviceId_AdrTmp[4]:=T_DeviceId.T_LightbusMaster;
		(* NovRAM name *)
		T_DeviceId_AdrTmp[3]:=T_DeviceId.T_NovRAM;
		(* end *)
		T_DeviceId_AdrTmp[5].sDeviceName:='';
		(*reset variable*)
		xInitReadStructure:=FALSE;
		iPtrDeviceName:=1;
		(* start device id reading *)
		xGetDeviceId:=TRUE;
	(* Exit FB *)
		RETURN;
	END_IF

(* get device Id *)
	IF xGetDeviceId THEN
		FallingEdgeBusy(CLK:=FBGeviceInfoByName.BUSY);
		IF FallingEdgeBusy.Q THEN
		(* save device id *)
			T_DeviceId_AdrTmp[iPtrDeviceName].udiDeviceID:=FBGeviceInfoByName.DEVICEID;
			T_DeviceId_AdrTmp[iPtrDeviceName].sAmsNetId:=FBGeviceInfoByName.DEVICENETID;
			(* next device *)
			iPtrDeviceName:=iPtrDeviceName+1;
		END_IF
		IF NOT(FBGeviceInfoByName.BUSY) AND T_DeviceId_AdrTmp[iPtrDeviceName].sDeviceName <> '' THEN
			FBGeviceInfoByName(	NETID:='',
								DEVICENAME:=T_DeviceId_AdrTmp[iPtrDeviceName].sDeviceName,
								START:=TRUE,
								TMOUT:=T#2s);
		ELSE
			FBGeviceInfoByName(START:=FALSE);
		END_IF
		IF NOT(FBGeviceInfoByName.BUSY) AND NOT(FBGeviceInfoByName.ERR) AND T_DeviceId_AdrTmp[iPtrDeviceName].sDeviceName = '' THEN
			(* init. variable *)
			xGetDeviceId:=FALSE;
			(* set copy value *)
			xCopyReadyStructure:=TRUE;
		END_IF
		IF FBGeviceInfoByName.ERR THEN
		(* acitve error *)
			IF NOT(T_DeviceId_AdrTmp[iPtrDeviceName].xDeviceOption) THEN
				IF (iPtrDeviceName <> 5) THEN
					ptrDeviceId^.T_Ctrle.xDone:=FALSE;
					ptrDeviceId^.T_Ctrle.xErr:=TRUE;
					ptrDeviceId^.T_Ctrle.udiErrorID:=FBGeviceInfoByName.ERRID;
					(* init. variable *)
					xGetDeviceId:=FALSE;
				ELSE
					(* init. variable *)
					xGetDeviceId:=FALSE;
					(* set copy value *)
					xCopyReadyStructure:=TRUE;
				END_IF;
			END_IF
		END_IF
	ELSE
		FBGeviceInfoByName(START:=FALSE);
	END_IF

(* copy read value *)
	IF xCopyReadyStructure THEN
	(* copy value *)
		(* PLC name *)
		T_DeviceId.T_CX1020:=T_DeviceId_AdrTmp[1];
		(* feldbus name *)
		T_DeviceId.T_CANOpenMaster:=T_DeviceId_AdrTmp[2];
		T_DeviceId.T_LightbusMaster:=T_DeviceId_AdrTmp[4];
		(* NovRAM name *)
		T_DeviceId.T_NovRAM:=T_DeviceId_AdrTmp[3];
		(* confirm device list id *)
		ptrDeviceId^.T_Ctrle.xDone:=TRUE;
		ptrDeviceId^.T_Ctrle.xErr:=FALSE;
		ptrDeviceId^.T_Ctrle.udiErrorID:=0;
		(* reset variable *)
		xCopyReadyStructure:=FALSE;
	END_IF
END_FUNCTION_BLOCK

(* POU FB_HARDWARE/FBHW_BOXID, ST *)
FUNCTION_BLOCK FBHW_BOXID
VAR_INPUT
	udiDeviceIdLightBusMaster:UDINT;
END_VAR
VAR_IN_OUT
	T_BoxId:ST_BOXID;
END_VAR
VAR_OUTPUT
END_VAR
VAR
(* pointer of Box ID *)
	ptrBoxId: POINTER TO ST_BOXID;
(* function bloc *)
	fbGetBoxAddrByName:IOF_GetBoxAddrByName;
	fbGetBoxNetId:IOF_GetBoxNetId;
(* trigger *)
	RisingEdgeResetFB:R_TRIG;
	RisingEdgeExecute:R_TRIG;
(* variable *)
	xGetBoxId:BOOL:=FALSE;
	xConfirmResetFB:BOOL:=FALSE;
	iPtrBoxName:INT:=0;
	iPtrBoxNameEnd:INT:=0;
	T_BoxId_AdrTmp:ARRAY[1..20] OF ST_BOXID_DATA_ADR;
	xInitReadStructure: BOOL;
	xCopyReadyStructure:BOOL;
	xGetBoxAddress: BOOL;
END_VAR
(****************************************************************************************************************************************************)
(***********                     This Functionblock is needed for read the BoxID information of the Beckhoff components               ************)
(****************************************************************************************************************************************************)
(* reset *)
	RisingEdgeResetFB(CLK:=T_BoxId.T_Ctrle.xReset);
	IF RisingEdgeResetFB.Q THEN
	(* init ptr*)
		ptrBoxId:=ADR(T_BoxId);
	(* init. variable *)
		xGetBoxId:=FALSE;
		iPtrBoxName:=1;
	(* Init. variable *)
		ptrBoxId^.T_Ctrle.xDone:=FALSE;
		ptrBoxId^.T_Ctrle.xErr:=FALSE;
		ptrBoxId^.T_Ctrle.udiErrorID:=0;
	(* activ confirm reset *)
		xConfirmResetFB:=TRUE;
	(* Exit FB *)
		RETURN;
	ELSE
		IF xConfirmResetFB THEN
		(* confirm reset FB *)
			ptrBoxId^.T_Ctrle.xDone:=TRUE;
			ptrBoxId^.T_Ctrle.xErr:=FALSE;
			ptrBoxId^.T_Ctrle.udiErrorID:=0;
		(* reset variable *)
			xConfirmResetFB:=FALSE;
		END_IF
	END_IF

(* execute *)
	RisingEdgeExecute(CLK:=T_BoxId.T_Ctrle.xExecute);
	IF RisingEdgeExecute.Q THEN
	(* init ptr*)
		ptrBoxId:=ADR(T_BoxId);
	(* activ get device Id *)
		xInitReadStructure:=TRUE;
	(* init. state flag *)
		ptrBoxId^.T_Ctrle.xDone:=FALSE;
		ptrBoxId^.T_Ctrle.xErr:=FALSE;
		ptrBoxId^.T_Ctrle.udiErrorID:=0;
	(* Exit FB *)
		RETURN;
	END_IF

(* init. read structure *)
	IF xInitReadStructure THEN
	(* PLC name, servo  *)
		iPtrBoxName:=1;
		T_BoxId_AdrTmp[1]:=T_BoxId.T_Servo_ToolLeft;
		T_BoxId_AdrTmp[2]:=T_BoxId.T_Servo_ToolCenter;
		T_BoxId_AdrTmp[3]:=T_BoxId.T_Servo_ToolRight;
		T_BoxId_AdrTmp[4]:=T_BoxId.T_Servo_ToolFeeder;
		T_BoxId_AdrTmp[5]:=T_BoxId.T_Servo_GrindFeeder;
		iPtrBoxNameEnd:=5;
		(* end *)
		T_BoxId_AdrTmp[6].sDeviceName:='';
		(*reset variable*)
		xInitReadStructure:=FALSE;
		(* start device id reading *)
		xGetBoxAddress:=TRUE;
	(* Exit FB *)
		RETURN;
	END_IF

(* get box address *)
	IF xGetBoxAddress THEN
		fbGetBoxAddrByName(	NETID:='',
								DEVICEID:=udiDeviceIdLightBusMaster,
								BOXNAME:=T_BoxId_AdrTmp[iPtrBoxName].sBoxName,
								START:=TRUE,
								TMOUT:=T#2s);
		IF NOT(fbGetBoxAddrByName.BUSY) OR fbGetBoxAddrByName.ERR THEN
			IF fbGetBoxAddrByName.ERR THEN
				IF T_BoxId_AdrTmp[iPtrBoxName].xDeviceOption THEN
				(* Init. FB *)
					fbGetBoxAddrByName(START:=FALSE);
					IF iPtrBoxName <> iPtrBoxNameEnd THEN
					(* next box *)
						iPtrBoxName:=iPtrBoxName+1;
						IF (T_BoxId.T_Ctrle.iMachineType = 1) AND (iPtrBoxName = 2) THEN
							iPtrBoxName:=3;
						END_IF;
						(* exit FB *)
						RETURN;
					(* activ copy value *)
					ELSE xCopyReadyStructure:=TRUE;END_IF
				ELSE
				(* acitve error *)
					ptrBoxId^.T_Ctrle.xDone:=FALSE;
					ptrBoxId^.T_Ctrle.xErr:=TRUE;
					ptrBoxId^.T_Ctrle.udiErrorID:=fbGetBoxAddrByName.ERRID;
				END_IF
			ELSE
			(* get address *)
				T_BoxId_AdrTmp[iPtrBoxName].wAddrBox:=UINT_TO_WORD(fbGetBoxAddrByName.BOXADDR);
				(* enable get box id *)
				xGetBoxId:=TRUE;
			END_IF
			(* disable get address *)
			xGetBoxAddress:=FALSE;
		END_IF
	ELSE
		fbGetBoxAddrByName(START:=FALSE);
	END_IF

(* get device Id *)
	IF xGetBoxId THEN
		fbGetBoxNetId(	NETID:='',
						DEVICEID:=udiDeviceIdLightBusMaster,
						BOXADDR:=T_BoxId_AdrTmp[iPtrBoxName].wAddrBox,
						START:=TRUE,
						TMOUT:=T#2s);
		IF NOT(fbGetBoxNetId.BUSY) OR fbGetBoxNetId.ERR THEN
			IF fbGetBoxNetId.ERR THEN
			(* acitve error *)
				ptrBoxId^.T_Ctrle.xDone:=FALSE;
				ptrBoxId^.T_Ctrle.xErr:=TRUE;
				ptrBoxId^.T_Ctrle.udiErrorID:=fbGetBoxNetId.ERRID;
			ELSE
				(* get BoxID *)
				T_BoxId_AdrTmp[iPtrBoxName].sAmsNetId:=fbGetBoxNetId.BoxNetId;
				IF iPtrBoxName <> iPtrBoxNameEnd THEN
				(* next box *)
					iPtrBoxName:=iPtrBoxName+1;
					IF (T_BoxId.T_Ctrle.iMachineType = 1) AND (iPtrBoxName = 2) THEN
						iPtrBoxName:=3;
					END_IF;
					(* activ get address *)
					xGetBoxAddress:=TRUE;
				ELSE
				(* activ copy value *)
					xCopyReadyStructure:=TRUE;
				END_IF
			END_IF
			(* init. variable *)
			xGetBoxId:=FALSE;
		END_IF
	ELSE
		fbGetBoxNetId(START:=FALSE);
	END_IF

(* copy read value *)
	IF xCopyReadyStructure THEN
	(* copy value *)
		T_BoxId.T_Servo_ToolLeft:=T_BoxId_AdrTmp[1];
		T_BoxId.T_Servo_ToolCenter:=T_BoxId_AdrTmp[2];
		T_BoxId.T_Servo_ToolRight:=T_BoxId_AdrTmp[3];
		T_BoxId.T_Servo_ToolFeeder:=T_BoxId_AdrTmp[4];
		T_BoxId.T_Servo_GrindFeeder:=T_BoxId_AdrTmp[5];
		(* confirm device list id *)
		ptrBoxId^.T_Ctrle.xDone:=TRUE;
		ptrBoxId^.T_Ctrle.xErr:=FALSE;
		ptrBoxId^.T_Ctrle.udiErrorID:=0;
		(* reset variable *)
		xCopyReadyStructure:=FALSE;
	END_IF
END_FUNCTION_BLOCK

(* POU PRG_VISU_LAYER5/FB_VISU/FB_PROFILE_FILE, ST *)
FUNCTION_BLOCK FB_PROFILE_FILE
VAR_INPUT
END_VAR
VAR_OUTPUT
END_VAR
VAR_IN_OUT
	T_Data_ProcessImageLoadData:ST_RETAIN_DATA_PROCESSIMAGE;		(* Novram parameter structure for the profile value *)
	T_Data_ProcessImageData:ST_RETAIN_DATA_PROCESSIMAGE;			(* Novram parametre structure for the process parameter *)
	T_Profile:ST_PROFILE;												(* data structure for the profile mangement *)
	T_HDD:ST_HDD;														(* data structure for the file managment *)
END_VAR
VAR
(* Timer *)
	TimerOut:TON;
(* Trigger *)
	RisingEdgeReset:R_TRIG;
	RisingEdgeExecute:R_TRIG;
(* variable *)
	xConfirmResetFB:BOOL;
	xReadProfile:BOOL;
	xWriteProfile:BOOL;
	xReadProfileListeStation: BOOL;
	iStepFunction:INT;
	xStepFunctionDone:BOOL;
	tTimeOut: TIME;
(* Tmp *)
	xTmp:BOOL;
	sTmp:STRING;
END_VAR
(****************************************************************************************************************************************************)
(***********                                       This Functionblock manage the profile for read and write to a file                                            ************)
(****************************************************************************************************************************************************)
(* waiting for reset *)
	RisingEdgeReset(CLK:=T_Profile.T_Ctrle.xReset);
	IF RisingEdgeReset.Q THEN
	(* init. structure *)
		T_Profile.T_Ctrle.xDone:=FALSE;
		T_Profile.T_Ctrle.xErr:=FALSE;
		T_Profile.T_Ctrle.udiErrorID:=0;
		T_Profile.T_Ctrle.iFunction:=0;
		(* Reset HDD if error activ *)
		IF T_HDD.T_Ctrle.xErr THEN T_HDD.T_Ctrle.xReset:=TRUE; END_IF
		(* Init. variable *)
		xReadProfile:=FALSE;
		xWriteProfile:=FALSE;
		xReadProfileListeStation:=FALSE;
		(* set flag done *)
		xConfirmResetFB:=TRUE;
		(* exit function *)
		RETURN;
	ELSE
		IF xConfirmResetFB THEN
		(* confirm reset FB *)
			T_Profile.T_Ctrle.xDone:=TRUE;
			T_Profile.T_Ctrle.xErr:=FALSE;
			T_Profile.T_Ctrle.udiErrorID:=0;
			T_Profile.T_Ctrle.iFunction:=0;
			(* init. variable *)
			xConfirmResetFB:=FALSE;
		END_IF
	END_IF

(* waiting for execute *)
	RisingEdgeExecute(CLK:=T_Profile.T_Ctrle.xExecute);
	IF RisingEdgeExecute.Q THEN
		CASE T_Profile.T_Ctrle.iFunction OF
		(* read profile *)
		1:	xReadProfile:=TRUE;
			tTimeOut:=T#5s;
		(* write profile *)
		2:	xWriteProfile:=TRUE;
			tTimeOut:=T#5s;
		(* read profile liste station *)
		3:	xReadProfileListeStation:=TRUE;
			tTimeOut:=T#20s;
		ELSE
		(* function not implemented *)
			 T_Profile.T_Ctrle.xDone:=FALSE;
			 T_Profile.T_Ctrle.xErr:=TRUE;
			 T_Profile.T_Ctrle.udiErrorID:=16#F000;
			 (* exit FB *)
			 RETURN;
		END_CASE
		(* Init. variable *)
		T_Profile.T_Ctrle.xDone:=FALSE;
		T_Profile.T_Ctrle.xErr:=FALSE;
		T_Profile.T_Ctrle.udiErrorID:=16#0;
		(* init. step *)
		iStepFunction:=1;
		xStepFunctionDone:=FALSE;
		RETURN;
	END_IF

(* Monitor time out *)
	xTmp:=	NOT T_Profile.T_Ctrle.xDone
			AND NOT T_Profile.T_Ctrle.xErr;
	TimerOut(IN:=xTmp, PT:=tTimeOut);
	IF TimerOut.Q THEN iStepFunction:=99; END_IF

(* Read profile *)
	IF xReadProfile OR xWriteProfile THEN
		CASE iStepFunction OF
		(* check if HDD state *)
		1:	xTmp:=	T_HDD.T_Ctrle.xDone
					AND NOT T_HDD.T_Ctrle.xExecute
					AND NOT T_HDD.T_Ctrle.xErr
					AND NOT T_HDD.T_Ctrle.xLocked;
			IF xTmp THEN iStepFunction:=10; ELSE iStepFunction:=95; END_IF
			IF T_HDD.T_Ctrle.xErr THEN iStepFunction:=99; END_IF
		(* file name and activ read *)
		10:	sTmp:='\Hard Disk\Machine450\Profile\';
			sTmp:=CONCAT(sTmp,T_Profile.T_Id.sName);
			IF xReadProfile THEN
			(* activ read *)
				T_HDD.T_Ctrle.iFunction:=1;
				T_HDD.T_File.sPathAndFileName:=CONCAT(sTmp,'.txt');
				T_HDD.T_Ctrle.xExecute:=TRUE;
				(* next step *)
				iStepFunction:=20;
				xStepFunctionDone:=FALSE;
			(* activ write *)
			ELSE
				(* copy profile to HDD data structure *)

				IF xFctCopyProfileToDataFile(	ptrData_ProcessImageData:=ADR(T_Data_ProcessImageData),
											ptrDataFile:=ADR(T_HDD.T_Data))	THEN iStepFunction:=50; ELSE iStepFunction:=99; END_IF;
				(* next step *)
				xStepFunctionDone:=FALSE;
			END_IF
		(* waiting flag *)
		20:	IF T_HDD.T_Ctrle.xDone THEN iStepFunction:=30; END_IF
			IF T_HDD.T_Ctrle.xErr THEN iStepFunction:=80; END_IF
		(* copy value from HDD to Profile structure *)
		30:	IF xFctCopyDataFileToProfile(	ptrData_ProcessImageLoadData:=ADR(T_Data_ProcessImageLoadData),
										ptrDataFile:=ADR(T_HDD.T_Data))	THEN iStepFunction:=90; ELSE iStepFunction:=99; END_IF;
		(* activ write *)
		50:	sTmp:='\Hard Disk\Machine450\Profile\';
			sTmp:=CONCAT(sTmp,T_Profile.T_Id.sName);
			T_HDD.T_File.sPathAndFileName:=CONCAT(sTmp,'.txt');
			T_HDD.T_Ctrle.iFunction:=2;
			T_HDD.T_Ctrle.xExecute:=TRUE;
			(* next step *)
			iStepFunction:=60;
			xStepFunctionDone:=FALSE;
		(* waiting flag *)
		60:	IF T_HDD.T_Ctrle.xDone THEN iStepFunction:=90; END_IF
			IF T_HDD.T_Ctrle.xErr THEN iStepFunction:=80; END_IF
		(* reset error *)
		80:	T_HDD.T_Ctrle.xReset:=TRUE;
			iStepFunction:=99;
		(* done *)
		90:	T_Profile.T_Ctrle.xDone:=TRUE;
			T_Profile.T_Ctrle.xErr:=FALSE;
			T_Profile.T_Ctrle.udiErrorID:=16#0;
			xReadProfile:=FALSE;
			xWriteProfile:=FALSE;
		(* not ready *)
		95:	T_Profile.T_Ctrle.xDone:=TRUE;
			T_Profile.T_Ctrle.xErr:=FALSE;
			T_Profile.T_Ctrle.udiErrorID:=16#0;
			xReadProfile:=FALSE;
			xWriteProfile:=FALSE;
		(* error *)
		99:	T_Profile.T_Ctrle.xDone:=FALSE;
			T_Profile.T_Ctrle.xErr:=TRUE;
			T_Profile.T_Ctrle.udiErrorID:=16#F1000 + T_Profile.T_Ctrle.iFunction;
			xReadProfile:=FALSE;
			xWriteProfile:=FALSE;
		END_CASE
	END_IF
END_FUNCTION_BLOCK

(* POU PRG_VISU_LAYER5/FB_VISU/xFctCopyProfileToDataFile, ST *)
FUNCTION xFctCopyProfileToDataFile : BOOL
VAR_INPUT
	ptrData_ProcessImageData:POINTER TO ST_RETAIN_DATA_PROCESSIMAGE;	(* Novram parametre structure for the process parameter *)
	ptrDataFile:POINTER TO ARRAY[1..csiMaxFileLine] OF STRING(255);				(* structure of the data file *)
END_VAR
VAR
(* variable *)
	i:INT;
(* Tmp *)
	sTmp:STRING;
END_VAR
(****************************************************************************************************************************************************)
(***********                     This Function make a copy from the profile structure to the readed profil parameter                           ************)
(****************************************************************************************************************************************************)
(* Init. variable *)
	xFctCopyProfileToDataFile:=FALSE;
	i:=1;
(* copy value *)
	ptrDataFile^[i]:='/* Geometry Section 1 */';i:=i+1;
	sTmp:=CONCAT('01:rStartDiameterS1:=',REAL_TO_STRING(ptrData_ProcessImageData^.T_GeometryPara.arStartDiameter[1]));
	ptrDataFile^[i]:=CONCAT(sTmp,';');i:=i+1;
	sTmp:=CONCAT('02:rEndDiameterS1:=',REAL_TO_STRING(ptrData_ProcessImageData^.T_GeometryPara.arEndDiameter[1]));
	ptrDataFile^[i]:=CONCAT(sTmp,';');i:=i+1;
	sTmp:=CONCAT('03:rLengthS1:=',REAL_TO_STRING(ptrData_ProcessImageData^.T_GeometryPara.arSectionLength[1]));
	ptrDataFile^[i]:=CONCAT(sTmp,';');i:=i+1;
	sTmp:=CONCAT('04:rPitchS1:=',REAL_TO_STRING(ptrData_ProcessImageData^.T_GeometryPara.arSectionPitch[1]));
	ptrDataFile^[i]:=CONCAT(sTmp,';');i:=i+1;
	IF ptrData_ProcessImageData^.T_GeometryPara.axActiveSection[1] THEN
		sTmp:=CONCAT('05:rActiveS1:=','1');
	ELSE
		sTmp:=CONCAT('05:rActiveS1:=','0');
	END_IF;
	ptrDataFile^[i]:=CONCAT(sTmp,';');i:=i+1;

	ptrDataFile^[i]:='/* Geometry Section 2 */';i:=i+1;
	sTmp:=CONCAT('06:rStartDiameterS2:=',REAL_TO_STRING(ptrData_ProcessImageData^.T_GeometryPara.arStartDiameter[2]));
	ptrDataFile^[i]:=CONCAT(sTmp,';');i:=i+1;
	sTmp:=CONCAT('07:rEndDiameterS2:=',REAL_TO_STRING(ptrData_ProcessImageData^.T_GeometryPara.arEndDiameter[2]));
	ptrDataFile^[i]:=CONCAT(sTmp,';');i:=i+1;
	sTmp:=CONCAT('08:rLengthS2:=',REAL_TO_STRING(ptrData_ProcessImageData^.T_GeometryPara.arSectionLength[2]));
	ptrDataFile^[i]:=CONCAT(sTmp,';');i:=i+1;
	sTmp:=CONCAT('09:rPitchS2:=',REAL_TO_STRING(ptrData_ProcessImageData^.T_GeometryPara.arSectionPitch[2]));
	ptrDataFile^[i]:=CONCAT(sTmp,';');i:=i+1;
	IF ptrData_ProcessImageData^.T_GeometryPara.axActiveSection[2] THEN
		sTmp:=CONCAT('10:rActiveS2:=','1');
	ELSE
		sTmp:=CONCAT('10:rActiveS2:=','0');
	END_IF;
	ptrDataFile^[i]:=CONCAT(sTmp,';');i:=i+1;

	ptrDataFile^[i]:='/* Geometry Section 3 */';i:=i+1;
	sTmp:=CONCAT('11:rStartDiameterS3:=',REAL_TO_STRING(ptrData_ProcessImageData^.T_GeometryPara.arStartDiameter[3]));
	ptrDataFile^[i]:=CONCAT(sTmp,';');i:=i+1;
	sTmp:=CONCAT('12:rEndDiameterS3:=',REAL_TO_STRING(ptrData_ProcessImageData^.T_GeometryPara.arEndDiameter[3]));
	ptrDataFile^[i]:=CONCAT(sTmp,';');i:=i+1;
	sTmp:=CONCAT('13:rLengthS3:=',REAL_TO_STRING(ptrData_ProcessImageData^.T_GeometryPara.arSectionLength[3]));
	ptrDataFile^[i]:=CONCAT(sTmp,';');i:=i+1;
	sTmp:=CONCAT('14:rPitchS3:=',REAL_TO_STRING(ptrData_ProcessImageData^.T_GeometryPara.arSectionPitch[3]));
	ptrDataFile^[i]:=CONCAT(sTmp,';');i:=i+1;
	IF ptrData_ProcessImageData^.T_GeometryPara.axActiveSection[3] THEN
		sTmp:=CONCAT('15:rActiveS3:=','1');
	ELSE
		sTmp:=CONCAT('15:rActiveS3:=','0');
	END_IF;
	ptrDataFile^[i]:=CONCAT(sTmp,';');i:=i+1;

	ptrDataFile^[i]:='/* Geometry Section 4 */';i:=i+1;
	sTmp:=CONCAT('16:rStartDiameterS4:=',REAL_TO_STRING(ptrData_ProcessImageData^.T_GeometryPara.arStartDiameter[4]));
	ptrDataFile^[i]:=CONCAT(sTmp,';');i:=i+1;
	sTmp:=CONCAT('17:rEndDiameterS4:=',REAL_TO_STRING(ptrData_ProcessImageData^.T_GeometryPara.arEndDiameter[4]));
	ptrDataFile^[i]:=CONCAT(sTmp,';');i:=i+1;
	sTmp:=CONCAT('18:rLengthS4:=',REAL_TO_STRING(ptrData_ProcessImageData^.T_GeometryPara.arSectionLength[4]));
	ptrDataFile^[i]:=CONCAT(sTmp,';');i:=i+1;
	sTmp:=CONCAT('19:rPitchS4:=',REAL_TO_STRING(ptrData_ProcessImageData^.T_GeometryPara.arSectionPitch[4]));
	ptrDataFile^[i]:=CONCAT(sTmp,';');i:=i+1;
	IF ptrData_ProcessImageData^.T_GeometryPara.axActiveSection[4] THEN
		sTmp:=CONCAT('20:rActiveS4:=','1');
	ELSE
		sTmp:=CONCAT('20:rActiveS4:=','0');
	END_IF;
	ptrDataFile^[i]:=CONCAT(sTmp,';');i:=i+1;
(*09.12.2022: SOA	{	 *)
	ptrDataFile^[i]:='/* Geometry Section 5 */';i:=i+1;
	sTmp:=CONCAT('21:rStartDiameterS5:=',REAL_TO_STRING(ptrData_ProcessImageData^.T_GeometryPara.arStartDiameter[5]));
	ptrDataFile^[i]:=CONCAT(sTmp,';');i:=i+1;
	sTmp:=CONCAT('22:rEndDiameterS5:=',REAL_TO_STRING(ptrData_ProcessImageData^.T_GeometryPara.arEndDiameter[5]));
	ptrDataFile^[i]:=CONCAT(sTmp,';');i:=i+1;
	sTmp:=CONCAT('23:rLengthS5:=',REAL_TO_STRING(ptrData_ProcessImageData^.T_GeometryPara.arSectionLength[5]));
	ptrDataFile^[i]:=CONCAT(sTmp,';');i:=i+1;
	sTmp:=CONCAT('24:rPitchS1:=',REAL_TO_STRING(ptrData_ProcessImageData^.T_GeometryPara.arSectionPitch[5]));
	ptrDataFile^[i]:=CONCAT(sTmp,';');i:=i+1;
	IF ptrData_ProcessImageData^.T_GeometryPara.axActiveSection[5] THEN
		sTmp:=CONCAT('25:rActiveS5:=','1');
	ELSE
		sTmp:=CONCAT('25:rActiveS5:=','0');
	END_IF;
	ptrDataFile^[i]:=CONCAT(sTmp,';');i:=i+1;

	ptrDataFile^[i]:='/* Geometry Section 6 */';i:=i+1;
	sTmp:=CONCAT('26:rStartDiameterS6:=',REAL_TO_STRING(ptrData_ProcessImageData^.T_GeometryPara.arStartDiameter[6]));
	ptrDataFile^[i]:=CONCAT(sTmp,';');i:=i+1;
	sTmp:=CONCAT('27:rEndDiameterS6:=',REAL_TO_STRING(ptrData_ProcessImageData^.T_GeometryPara.arEndDiameter[6]));
	ptrDataFile^[i]:=CONCAT(sTmp,';');i:=i+1;
	sTmp:=CONCAT('28:rLengthS6:=',REAL_TO_STRING(ptrData_ProcessImageData^.T_GeometryPara.arSectionLength[6]));
	ptrDataFile^[i]:=CONCAT(sTmp,';');i:=i+1;
	sTmp:=CONCAT('29:rPitchS6:=',REAL_TO_STRING(ptrData_ProcessImageData^.T_GeometryPara.arSectionPitch[6]));
	ptrDataFile^[i]:=CONCAT(sTmp,';');i:=i+1;
	IF ptrData_ProcessImageData^.T_GeometryPara.axActiveSection[6] THEN
		sTmp:=CONCAT('30:rActiveS6:=','1');
	ELSE
		sTmp:=CONCAT('30:rActiveS6:=','0');
	END_IF;
(*09.12.2022: SOA	}	 *)
	ptrDataFile^[i]:=CONCAT(sTmp,';');i:=i+1;

	ptrDataFile^[i]:='/* Prism Parameter */';i:=i+1;
	sTmp:=CONCAT('31:rPrismaDistanceD1:=',REAL_TO_STRING(ptrData_ProcessImageData^.T_PrismPara.rPrismaDistanceD1));
	ptrDataFile^[i]:=CONCAT(sTmp,';');i:=i+1;
	sTmp:=CONCAT('32:rPrismaDistanceD2:=',REAL_TO_STRING(ptrData_ProcessImageData^.T_PrismPara.rPrismaDistanceD2));
	ptrDataFile^[i]:=CONCAT(sTmp,';');i:=i+1;
	sTmp:=CONCAT('33:rPrismaAngleA:=',REAL_TO_STRING(ptrData_ProcessImageData^.T_PrismPara.rPrismaAngleA));
	ptrDataFile^[i]:=CONCAT(sTmp,';');i:=i+1;
	sTmp:=CONCAT('34:bStateInputPrisma:=',BYTE_TO_STRING(ptrData_ProcessImageData^.T_PrismPara.bStateInputPrisma));
	ptrDataFile^[i]:=CONCAT(sTmp,';');i:=i+1;
	sTmp:=CONCAT('35:rToolDiameterMin:=',REAL_TO_STRING(ptrData_ProcessImageData^.T_PrismPara.rToolDiameterMin));
	ptrDataFile^[i]:=CONCAT(sTmp,';');i:=i+1;
	sTmp:=CONCAT('36:rToolDiameterMax:=',REAL_TO_STRING(ptrData_ProcessImageData^.T_PrismPara.rToolDiameterMax));
	ptrDataFile^[i]:=CONCAT(sTmp,';');i:=i+1;
	sTmp:=CONCAT('37:rPrismaFactor:=',REAL_TO_STRING(ptrData_ProcessImageData^.T_PrismPara.rPrismaFactor));
	ptrDataFile^[i]:=CONCAT(sTmp,';');i:=i+1;

	ptrDataFile^[i]:='/* Auto Geometry */';i:=i+1;
	sTmp:=CONCAT('38:iCycleGeometry:=',INT_TO_STRING(ptrData_ProcessImageData^.T_AutoGeometryPara.iCycleGeometry));
	ptrDataFile^[i]:=CONCAT(sTmp,';');i:=i+1;
	sTmp:=CONCAT('39:rPlungeCycleGrindFeedGeometry:=',REAL_TO_STRING(ptrData_ProcessImageData^.T_AutoGeometryPara.rPlungeCycleGrindFeedGeometry));
	ptrDataFile^[i]:=CONCAT(sTmp,';');i:=i+1;
	sTmp:=CONCAT('40:rDisplaceLengthToolFeedGeometry:=',REAL_TO_STRING(ptrData_ProcessImageData^.T_AutoGeometryPara.rDisplaceLengthToolFeedGeometry));
	ptrDataFile^[i]:=CONCAT(sTmp,';');i:=i+1;
	sTmp:=CONCAT('41:rDisplaceSpeedGrindFeedGeometry:=',REAL_TO_STRING(ptrData_ProcessImageData^.T_AutoGeometryPara.rDisplaceSpeedGrindFeedGeometry));
	ptrDataFile^[i]:=CONCAT(sTmp,';');i:=i+1;
	sTmp:=CONCAT('42:rPlungeLengthToolFeedGeometry:=',REAL_TO_STRING(ptrData_ProcessImageData^.T_AutoGeometryPara.rPlungeLengthToolFeedGeometry));
	ptrDataFile^[i]:=CONCAT(sTmp,';');i:=i+1;
	sTmp:=CONCAT('43:rPlungeSpeedGrindFeedGeometry:=',REAL_TO_STRING(ptrData_ProcessImageData^.T_AutoGeometryPara.rPlungeSpeedGrindFeedGeometry));
	ptrDataFile^[i]:=CONCAT(sTmp,';');i:=i+1;
	sTmp:=CONCAT('44:rSpeedToolRotationGeometry:=',REAL_TO_STRING(ptrData_ProcessImageData^.T_AutoGeometryPara.rSpeedToolRotationGeometry));
	ptrDataFile^[i]:=CONCAT(sTmp,';');i:=i+1;
	IF ptrData_ProcessImageData^.T_AutoGeometryPara.xDisplaceActivationGeometry THEN
		sTmp:=CONCAT('45:rDisplaceActivationGeometry:=','1');
	ELSE
		sTmp:=CONCAT('45:rDisplaceActivationGeometry:=','0');
	END_IF;
	ptrDataFile^[i]:=CONCAT(sTmp,';');i:=i+1;
	IF ptrData_ProcessImageData^.T_AutoGeometryPara.xPlungeActivationGeometry THEN
		sTmp:=CONCAT('46:rPlungeActivationGeometry:=','1');
	ELSE
		sTmp:=CONCAT('46:rPlungeActivationGeometry:=','0');
	END_IF;
	ptrDataFile^[i]:=CONCAT(sTmp,';');i:=i+1;

	ptrDataFile^[i]:='/* Auto Groove */';i:=i+1;
	sTmp:=CONCAT('47:rDisplaceLengthToolFeedGroove:=',REAL_TO_STRING(ptrData_ProcessImageData^.T_AutoGroovePara.rDisplaceLengthToolFeedGroove));
	ptrDataFile^[i]:=CONCAT(sTmp,';');i:=i+1;
	sTmp:=CONCAT('48:rDisplaceSpeedGrindFeedGroove:=',REAL_TO_STRING(ptrData_ProcessImageData^.T_AutoGroovePara.rDisplaceSpeedGrindFeedGroove));
	ptrDataFile^[i]:=CONCAT(sTmp,';');i:=i+1;
	sTmp:=CONCAT('49:rPitchGroove:=',REAL_TO_STRING(ptrData_ProcessImageData^.T_AutoGroovePara.rPitchGroove));
	ptrDataFile^[i]:=CONCAT(sTmp,';');i:=i+1;
	sTmp:=CONCAT('50:rPlungeLengthToolFeedGroove:=',REAL_TO_STRING(ptrData_ProcessImageData^.T_AutoGroovePara.rPlungeLengthToolFeedGroove));
	ptrDataFile^[i]:=CONCAT(sTmp,';');i:=i+1;
	sTmp:=CONCAT('51:rPlungeSpeedGrindFeedGroove:=',REAL_TO_STRING(ptrData_ProcessImageData^.T_AutoGroovePara.rPlungeSpeedGrindFeedGroove));
	ptrDataFile^[i]:=CONCAT(sTmp,';');i:=i+1;
	sTmp:=CONCAT('52:rSpeedToolRotationGroove:=',REAL_TO_STRING(ptrData_ProcessImageData^.T_AutoGroovePara.rSpeedToolRotationGroove));
	ptrDataFile^[i]:=CONCAT(sTmp,';');i:=i+1;
(*20091207*)
	sTmp:=CONCAT('53:iNumberOfGrooves:=',INT_TO_STRING(ptrData_ProcessImageData^.T_AutoGroovePara.iNumberOfGrooves));
	ptrDataFile^[i]:=CONCAT(sTmp,';');i:=i+1;

	IF ptrData_ProcessImageData^.T_AutoGroovePara.xDisplaceActivationGroove THEN
		sTmp:=CONCAT('54:rDisplaceActivationGroove:=','1');
	ELSE
		sTmp:=CONCAT('54:rDisplaceActivationGroove:=','0');
	END_IF;
	ptrDataFile^[i]:=CONCAT(sTmp,';');i:=i+1;
	IF ptrData_ProcessImageData^.T_AutoGroovePara.xPlungeActivationGroove THEN
		sTmp:=CONCAT('55:rPlungeActivationGroove:=','1');
	ELSE
		sTmp:=CONCAT('55:rPlungeActivationGroove:=','0');
	END_IF;
	ptrDataFile^[i]:=CONCAT(sTmp,';');i:=i+1;
	IF ptrData_ProcessImageData^.T_AutoGroovePara.xBlockGrindFeeder THEN
		sTmp:=CONCAT('56:rBlockGrindFeeder:=','1');
	ELSE
		sTmp:=CONCAT('56:rBlockGrindFeeder:=','0');
	END_IF;
	ptrDataFile^[i]:=CONCAT(sTmp,';');i:=i+1;

	ptrDataFile^[i]:='/* Calibration */';i:=i+1;
	sTmp:=CONCAT('57:rDisplaceLengthToolFeedCalib:=',REAL_TO_STRING(ptrData_ProcessImageData^.T_CalibrationPara.rDisplaceLengthToolFeedCalib));
	ptrDataFile^[i]:=CONCAT(sTmp,';');i:=i+1;
	sTmp:=CONCAT('58:rDisplaceSpeedGrindFeedCalib:=',REAL_TO_STRING(ptrData_ProcessImageData^.T_CalibrationPara.rDisplaceSpeedGrindFeedCalib));
	ptrDataFile^[i]:=CONCAT(sTmp,';');i:=i+1;
	sTmp:=CONCAT('59:rMeasureOffsetToolFeedCalib:=',REAL_TO_STRING(ptrData_ProcessImageData^.T_CalibrationPara.rMeasureOffsetToolFeedCalib));
	ptrDataFile^[i]:=CONCAT(sTmp,';');i:=i+1;
	sTmp:=CONCAT('60:rMeasurePosToolFeedCalib:=',REAL_TO_STRING(ptrData_ProcessImageData^.T_CalibrationPara.rMeasurePosToolFeedCalib));
	ptrDataFile^[i]:=CONCAT(sTmp,';');i:=i+1;
	sTmp:=CONCAT('61:rPitchCalib:=',REAL_TO_STRING(ptrData_ProcessImageData^.T_CalibrationPara.rPitchCalib));
	ptrDataFile^[i]:=CONCAT(sTmp,';');i:=i+1;
	sTmp:=CONCAT('62:rPlungeLengthGrindFeedCalib:=',REAL_TO_STRING(ptrData_ProcessImageData^.T_CalibrationPara.rPlungeLengthGrindFeedCalib));
	ptrDataFile^[i]:=CONCAT(sTmp,';');i:=i+1;
	sTmp:=CONCAT('63:rPlungeLengthToolFeedCalib:=',REAL_TO_STRING(ptrData_ProcessImageData^.T_CalibrationPara.rPlungeLengthToolFeedCalib));
	ptrDataFile^[i]:=CONCAT(sTmp,';');i:=i+1;
	sTmp:=CONCAT('64:rPlungeSpeedGrindFeedCalib:=',REAL_TO_STRING(ptrData_ProcessImageData^.T_CalibrationPara.rPlungeSpeedGrindFeedCalib));
	ptrDataFile^[i]:=CONCAT(sTmp,';');i:=i+1;
	sTmp:=CONCAT('65:rSpeedToolRotationCalib:=',REAL_TO_STRING(ptrData_ProcessImageData^.T_CalibrationPara.rSpeedToolRotationCalib));
	ptrDataFile^[i]:=CONCAT(sTmp,';');i:=i+1;
	sTmp:=CONCAT('66:rStartPosToolFeedCalib:=',REAL_TO_STRING(ptrData_ProcessImageData^.T_CalibrationPara.rStartPosToolFeedCalib));
	ptrDataFile^[i]:=CONCAT(sTmp,';');i:=i+1;
	sTmp:=CONCAT('67:rToolLengthCylinderPartCalib:=',REAL_TO_STRING(ptrData_ProcessImageData^.T_CalibrationPara.rToolLengthCylinderPartCalib));
	ptrDataFile^[i]:=CONCAT(sTmp,';');i:=i+1;
	IF ptrData_ProcessImageData^.T_CalibrationPara.xDisplaceActivationCalib THEN
		sTmp:=CONCAT('68:rDisplaceActivationCalib:=','1');
	ELSE
		sTmp:=CONCAT('58:rDisplaceActivationCalib:=','0');
	END_IF;
	ptrDataFile^[i]:=CONCAT(sTmp,';');i:=i+1;
	IF ptrData_ProcessImageData^.T_CalibrationPara.xPlungeActivationCalib THEN
		sTmp:=CONCAT('69:rPlungeActivationCalib:=','1');
	ELSE
		sTmp:=CONCAT('69:rPlungeActivationCalib:=','0');
	END_IF;
	ptrDataFile^[i]:=CONCAT(sTmp,';');i:=i+1;

	ptrDataFile^[i]:='/* Process Para */';i:=i+1;
	sTmp:=CONCAT('70:rOffsetBeforeToolDiaGrindFeedProcess:=',REAL_TO_STRING(ptrData_ProcessImageData^.T_ProcessPara.rOffsetBeforeToolDiaGrindFeedProcess));
	ptrDataFile^[i]:=CONCAT(sTmp,';');i:=i+1;
	sTmp:=CONCAT('71:rSecurityPosGrindFeedProcess:=',REAL_TO_STRING(ptrData_ProcessImageData^.T_ProcessPara.rSecurityPosGrindFeedProcess));
	ptrDataFile^[i]:=CONCAT(sTmp,';');i:=i+1;
	sTmp:=CONCAT('72:rSpeedBackwardGrindFeed:=',REAL_TO_STRING(ptrData_ProcessImageData^.T_ProcessPara.rSpeedBackwardGrindFeed));
	ptrDataFile^[i]:=CONCAT(sTmp,';');i:=i+1;
	sTmp:=CONCAT('73:rSpeedForwardFastGrindFeed:=',REAL_TO_STRING(ptrData_ProcessImageData^.T_ProcessPara.rSpeedForwardFastGrindFeed));
	ptrDataFile^[i]:=CONCAT(sTmp,';');i:=i+1;
	sTmp:=CONCAT('74:rSpeedForwardSlowGrindFeed:=',REAL_TO_STRING(ptrData_ProcessImageData^.T_ProcessPara.rSpeedForwardSlowGrindFeed));
	ptrDataFile^[i]:=CONCAT(sTmp,';');i:=i+1;
	sTmp:=CONCAT('75:rSpeedStartPosToolFeedProcess:=',REAL_TO_STRING(ptrData_ProcessImageData^.T_ProcessPara.rSpeedStartPosToolFeedProcess));
	ptrDataFile^[i]:=CONCAT(sTmp,';');i:=i+1;
	sTmp:=CONCAT('76:rStartPosToolFeedAuto:=',REAL_TO_STRING(ptrData_ProcessImageData^.T_ProcessPara.rStartPosToolFeedAuto));
	ptrDataFile^[i]:=CONCAT(sTmp,';');i:=i+1;
	sTmp:=CONCAT('77:rToolDiameterProcess:=',REAL_TO_STRING(ptrData_ProcessImageData^.T_ProcessPara.rToolDiameterProcess));
	ptrDataFile^[i]:=CONCAT(sTmp,';');i:=i+1;
	sTmp:=CONCAT('78:rToolTensionProcess:=',REAL_TO_STRING(ptrData_ProcessImageData^.T_ProcessPara.rToolTensionProcess));
	ptrDataFile^[i]:=CONCAT(sTmp,';');i:=i+1;

	(* add empty line to set the end *)
	ptrDataFile^[i]:='';

	(* confirm copy *)
	xFctCopyProfileToDataFile:=TRUE;
END_FUNCTION

(* POU PRG_VISU_LAYER5/FB_VISU/xFctCopyDataFileToProfile, ST *)
FUNCTION xFctCopyDataFileToProfile : BOOL
VAR_INPUT
	ptrData_ProcessImageLoadData:POINTER TO ST_RETAIN_DATA_PROCESSIMAGE;	(* Novram parameter structure for the profile value *)
	ptrDataFile:POINTER TO ARRAY[1..csiMaxFileLine] OF STRING(255);					(* structure of the data file *)
END_VAR
VAR
(* variable *)
	i:INT;
	iPosStartCarValue:INT;
	iPosStopCarValue:INT;
	sValue:STRING;
	sVariableName:STRING;
(* Tmp variable *)
	sTmp:STRING;
END_VAR
(****************************************************************************************************************************************************)
(***********                     This Function make a copy from the readed profil parameter to the profile structure                           ************)
(****************************************************************************************************************************************************)
(* Init. variable *)
	xFctCopyDataFileToProfile:=FALSE;

(* copy value *)
	FOR i:= 1 TO csiMaxFileLine DO
		sTmp:=ptrDataFile^[i];
		IF FIND(sTmp,':=') <> 0 THEN
		(* read value *)
			iPosStartCarValue:= FIND(sTmp,':=')+2;
			iPosStopCarValue:= FIND(sTmp,';');
			sValue:=MID(sTmp,iPosStopCarValue - iPosStartCarValue,iPosStartCarValue);
		(* read variable name *)
			iPosStartCarValue:= FIND(sTmp,':')+1;
			iPosStopCarValue:= FIND(sTmp,':=');
			sVariableName:=FCT_UPLOW_CASE(	xLowConvert:=TRUE,
												sInString:=MID(sTmp,iPosStopCarValue - iPosStartCarValue,iPosStartCarValue));
			(* Value *)
				IF sVariableName = 'rstartdiameters1' THEN ptrData_ProcessImageLoadData^.T_GeometryPara.arStartDiameter[1]:=STRING_TO_REAL(sValue); END_IF;
				IF sVariableName = 'renddiameters1' THEN ptrData_ProcessImageLoadData^.T_GeometryPara.arEndDiameter[1]:=STRING_TO_REAL(sValue); END_IF;
				IF sVariableName = 'rlengths1' THEN ptrData_ProcessImageLoadData^.T_GeometryPara.arSectionLength[1]:=STRING_TO_REAL(sValue); END_IF;
				IF sVariableName = 'rpitchs1' THEN ptrData_ProcessImageLoadData^.T_GeometryPara.arSectionPitch[1]:=STRING_TO_REAL(sValue); END_IF;
				IF sVariableName = 'ractives1' THEN
					IF (STRING_TO_REAL(sValue) = 0) THEN
						ptrData_ProcessImageLoadData^.T_GeometryPara.axActiveSection[1]:=FALSE;
					ELSE
						ptrData_ProcessImageLoadData^.T_GeometryPara.axActiveSection[1]:=TRUE;
					END_IF;
				END_IF;
				IF sVariableName = 'rstartdiameters2' THEN ptrData_ProcessImageLoadData^.T_GeometryPara.arStartDiameter[2]:=STRING_TO_REAL(sValue); END_IF;
				IF sVariableName = 'renddiameters2' THEN ptrData_ProcessImageLoadData^.T_GeometryPara.arEndDiameter[2]:=STRING_TO_REAL(sValue); END_IF;
				IF sVariableName = 'rlengths2' THEN ptrData_ProcessImageLoadData^.T_GeometryPara.arSectionLength[2]:=STRING_TO_REAL(sValue); END_IF;
				IF sVariableName = 'rpitchs2' THEN ptrData_ProcessImageLoadData^.T_GeometryPara.arSectionPitch[2]:=STRING_TO_REAL(sValue); END_IF;
				IF sVariableName = 'ractives2' THEN
					IF (STRING_TO_REAL(sValue) = 0) THEN
						ptrData_ProcessImageLoadData^.T_GeometryPara.axActiveSection[2]:=FALSE;
					ELSE
						ptrData_ProcessImageLoadData^.T_GeometryPara.axActiveSection[2]:=TRUE;
					END_IF;
				END_IF;
				IF sVariableName = 'rstartdiameters3' THEN ptrData_ProcessImageLoadData^.T_GeometryPara.arStartDiameter[3]:=STRING_TO_REAL(sValue); END_IF;
				IF sVariableName = 'renddiameters3' THEN ptrData_ProcessImageLoadData^.T_GeometryPara.arEndDiameter[3]:=STRING_TO_REAL(sValue); END_IF;
				IF sVariableName = 'rlengths3' THEN ptrData_ProcessImageLoadData^.T_GeometryPara.arSectionLength[3]:=STRING_TO_REAL(sValue); END_IF;
				IF sVariableName = 'rpitchs3' THEN ptrData_ProcessImageLoadData^.T_GeometryPara.arSectionPitch[3]:=STRING_TO_REAL(sValue); END_IF;
				IF sVariableName = 'ractives3' THEN
					IF (STRING_TO_REAL(sValue) = 0) THEN
						ptrData_ProcessImageLoadData^.T_GeometryPara.axActiveSection[3]:=FALSE;
					ELSE
						ptrData_ProcessImageLoadData^.T_GeometryPara.axActiveSection[3]:=TRUE;
					END_IF;
				END_IF;
				IF sVariableName = 'rstartdiameters4' THEN ptrData_ProcessImageLoadData^.T_GeometryPara.arStartDiameter[4]:=STRING_TO_REAL(sValue); END_IF;
				IF sVariableName = 'renddiameters4' THEN ptrData_ProcessImageLoadData^.T_GeometryPara.arEndDiameter[4]:=STRING_TO_REAL(sValue); END_IF;
				IF sVariableName = 'rlengths4' THEN ptrData_ProcessImageLoadData^.T_GeometryPara.arSectionLength[4]:=STRING_TO_REAL(sValue); END_IF;
				IF sVariableName = 'rpitchs4' THEN ptrData_ProcessImageLoadData^.T_GeometryPara.arSectionPitch[4]:=STRING_TO_REAL(sValue); END_IF;
				IF sVariableName = 'ractives4' THEN
					IF (STRING_TO_REAL(sValue) = 0) THEN
						ptrData_ProcessImageLoadData^.T_GeometryPara.axActiveSection[4]:=FALSE;
					ELSE
						ptrData_ProcessImageLoadData^.T_GeometryPara.axActiveSection[4]:=TRUE;
					END_IF;
				END_IF;
(*09.12.2022: SOA *)
				IF sVariableName = 'rstartdiameters5' THEN ptrData_ProcessImageLoadData^.T_GeometryPara.arStartDiameter[5]:=STRING_TO_REAL(sValue); END_IF;
				IF sVariableName = 'renddiameters5' THEN ptrData_ProcessImageLoadData^.T_GeometryPara.arEndDiameter[5]:=STRING_TO_REAL(sValue); END_IF;
				IF sVariableName = 'rlengths5' THEN ptrData_ProcessImageLoadData^.T_GeometryPara.arSectionLength[5]:=STRING_TO_REAL(sValue); END_IF;
				IF sVariableName = 'rpitchs5' THEN ptrData_ProcessImageLoadData^.T_GeometryPara.arSectionPitch[5]:=STRING_TO_REAL(sValue); END_IF;
				IF sVariableName = 'ractives5' THEN
					IF (STRING_TO_REAL(sValue) = 0) THEN
						ptrData_ProcessImageLoadData^.T_GeometryPara.axActiveSection[5]:=FALSE;
					ELSE
						ptrData_ProcessImageLoadData^.T_GeometryPara.axActiveSection[5]:=TRUE;
					END_IF;
				END_IF;
				IF sVariableName = 'rstartdiameters6' THEN ptrData_ProcessImageLoadData^.T_GeometryPara.arStartDiameter[6]:=STRING_TO_REAL(sValue); END_IF;
				IF sVariableName = 'renddiameters6' THEN ptrData_ProcessImageLoadData^.T_GeometryPara.arEndDiameter[6]:=STRING_TO_REAL(sValue); END_IF;
				IF sVariableName = 'rlengths6' THEN ptrData_ProcessImageLoadData^.T_GeometryPara.arSectionLength[6]:=STRING_TO_REAL(sValue); END_IF;
				IF sVariableName = 'rpitchs6' THEN ptrData_ProcessImageLoadData^.T_GeometryPara.arSectionPitch[6]:=STRING_TO_REAL(sValue); END_IF;
				IF sVariableName = 'ractives6' THEN
					IF (STRING_TO_REAL(sValue) = 0) THEN
						ptrData_ProcessImageLoadData^.T_GeometryPara.axActiveSection[6]:=FALSE;
					ELSE
						ptrData_ProcessImageLoadData^.T_GeometryPara.axActiveSection[6]:=TRUE;
					END_IF;
				END_IF;
(*09.12.2022: SOA *)

				IF sVariableName = 'rprismadistanced1' THEN ptrData_ProcessImageLoadData^.T_PrismPara.rPrismaDistanceD1:=STRING_TO_REAL(sValue); END_IF;
				IF sVariableName = 'rprismadistanced2' THEN ptrData_ProcessImageLoadData^.T_PrismPara.rPrismaDistanceD2:=STRING_TO_REAL(sValue); END_IF;
				IF sVariableName = 'rprismaanglea' THEN ptrData_ProcessImageLoadData^.T_PrismPara.rPrismaAngleA:=STRING_TO_REAL(sValue); END_IF;
				IF sVariableName = 'bstateinputprisma' THEN ptrData_ProcessImageLoadData^.T_PrismPara.bStateInputPrisma:=STRING_TO_BYTE(sValue); END_IF;
				IF sVariableName = 'rtooldiametermin' THEN ptrData_ProcessImageLoadData^.T_PrismPara.rToolDiameterMin:=STRING_TO_REAL(sValue); END_IF;
				IF sVariableName = 'rtooldiametermax' THEN ptrData_ProcessImageLoadData^.T_PrismPara.rToolDiameterMax:=STRING_TO_REAL(sValue); END_IF;
				IF sVariableName = 'rprismafactor' THEN ptrData_ProcessImageLoadData^.T_PrismPara.rPrismaFactor:=STRING_TO_REAL(sValue); END_IF;
				IF sVariableName = 'icyclegeometry' THEN ptrData_ProcessImageLoadData^.T_AutoGeometryPara.iCycleGeometry:=STRING_TO_INT(sValue); END_IF;
				IF sVariableName = 'rplungecyclegrindfeedgeometry' THEN ptrData_ProcessImageLoadData^.T_AutoGeometryPara.rPlungeCycleGrindFeedGeometry:=STRING_TO_REAL(sValue); END_IF;
				IF sVariableName = 'rdisplacelengthtoolfeedgeometry' THEN ptrData_ProcessImageLoadData^.T_AutoGeometryPara.rDisplaceLengthToolFeedGeometry:=STRING_TO_REAL(sValue); END_IF;
				IF sVariableName = 'rdisplacespeedgrindfeedgeometry' THEN ptrData_ProcessImageLoadData^.T_AutoGeometryPara.rDisplaceSpeedGrindFeedGeometry:=STRING_TO_REAL(sValue); END_IF;
				IF sVariableName = 'rplungelengthtoolfeedgeometry' THEN ptrData_ProcessImageLoadData^.T_AutoGeometryPara.rPlungeLengthToolFeedGeometry:=STRING_TO_REAL(sValue); END_IF;
				IF sVariableName = 'rplungespeedgrindfeedgeometry' THEN ptrData_ProcessImageLoadData^.T_AutoGeometryPara.rPlungeSpeedGrindFeedGeometry:=STRING_TO_REAL(sValue); END_IF;
				IF sVariableName = 'rspeedtoolrotationgeometry' THEN ptrData_ProcessImageLoadData^.T_AutoGeometryPara.rSpeedToolRotationGeometry:=STRING_TO_REAL(sValue); END_IF;
				IF sVariableName = 'rdisplaceactivationgeometry' THEN
					IF (STRING_TO_REAL(sValue) = 0) THEN
						ptrData_ProcessImageLoadData^.T_AutoGeometryPara.xDisplaceActivationGeometry:=FALSE;
					ELSE
						ptrData_ProcessImageLoadData^.T_AutoGeometryPara.xDisplaceActivationGeometry:=TRUE;
					END_IF;
				END_IF;
				IF sVariableName = 'rplungeactivationgeometry' THEN
					IF (STRING_TO_REAL(sValue) = 0) THEN
						ptrData_ProcessImageLoadData^.T_AutoGeometryPara.xPlungeActivationGeometry:=FALSE;
					ELSE
						ptrData_ProcessImageLoadData^.T_AutoGeometryPara.xPlungeActivationGeometry:=TRUE;
					END_IF;
				END_IF;
				IF sVariableName = 'rdisplacelengthtoolfeedgroove' THEN ptrData_ProcessImageLoadData^.T_AutoGroovePara.rDisplaceLengthToolFeedGroove:=STRING_TO_REAL(sValue); END_IF;
				IF sVariableName = 'rdisplacespeedgrindfeedgroove' THEN ptrData_ProcessImageLoadData^.T_AutoGroovePara.rDisplaceSpeedGrindFeedGroove:=STRING_TO_REAL(sValue); END_IF;
				IF sVariableName = 'rpitchgroove' THEN ptrData_ProcessImageLoadData^.T_AutoGroovePara.rPitchGroove:=STRING_TO_REAL(sValue); END_IF;
				IF sVariableName = 'rplungelengthtoolfeedgroove' THEN ptrData_ProcessImageLoadData^.T_AutoGroovePara.rPlungeLengthToolFeedGroove:=STRING_TO_REAL(sValue); END_IF;
				IF sVariableName = 'rplungespeedgrindfeedgroove' THEN ptrData_ProcessImageLoadData^.T_AutoGroovePara.rPlungeSpeedGrindFeedGroove:=STRING_TO_REAL(sValue); END_IF;
				IF sVariableName = 'rspeedtoolrotationgroove' THEN ptrData_ProcessImageLoadData^.T_AutoGroovePara.rSpeedToolRotationGroove:=STRING_TO_REAL(sValue); END_IF;
				IF sVariableName = 'inumberofgrooves' THEN ptrData_ProcessImageLoadData^.T_AutoGroovePara.iNumberOfGrooves:=STRING_TO_INT(sValue); END_IF;
				IF sVariableName = 'rdisplaceactivationgroove' THEN
					IF (STRING_TO_REAL(sValue) = 0) THEN
						ptrData_ProcessImageLoadData^.T_AutoGroovePara.xDisplaceActivationGroove:=FALSE;
					ELSE
						ptrData_ProcessImageLoadData^.T_AutoGroovePara.xDisplaceActivationGroove:=TRUE;
					END_IF;
				END_IF;
				IF sVariableName = 'rplungeactivationgroove' THEN
					IF (STRING_TO_REAL(sValue) = 0) THEN
						ptrData_ProcessImageLoadData^.T_AutoGroovePara.xPlungeActivationGroove:=FALSE;
					ELSE
						ptrData_ProcessImageLoadData^.T_AutoGroovePara.xPlungeActivationGroove:=TRUE;
					END_IF;
				END_IF;
				IF sVariableName = 'rblockgrindfeeder' THEN
					IF (STRING_TO_REAL(sValue) = 0) THEN
						ptrData_ProcessImageLoadData^.T_AutoGroovePara.xBlockGrindFeeder:=FALSE;
					ELSE
						ptrData_ProcessImageLoadData^.T_AutoGroovePara.xBlockGrindFeeder:=TRUE;
					END_IF;
				END_IF;
				IF sVariableName = 'rdisplacelengthtoolfeedcalib' THEN ptrData_ProcessImageLoadData^.T_CalibrationPara.rDisplaceLengthToolFeedCalib:=STRING_TO_REAL(sValue); END_IF;
				IF sVariableName = 'rdisplacespeedgrindfeedcalib' THEN ptrData_ProcessImageLoadData^.T_CalibrationPara.rDisplaceSpeedGrindFeedCalib:=STRING_TO_REAL(sValue); END_IF;
				IF sVariableName = 'rmeasureoffsettoolfeedcalib' THEN ptrData_ProcessImageLoadData^.T_CalibrationPara.rMeasureOffsetToolFeedCalib:=STRING_TO_REAL(sValue); END_IF;
				IF sVariableName = 'rmeasurepostoolfeedcalib' THEN ptrData_ProcessImageLoadData^.T_CalibrationPara.rMeasurePosToolFeedCalib:=STRING_TO_REAL(sValue); END_IF;
				IF sVariableName = 'rpitchcalib' THEN ptrData_ProcessImageLoadData^.T_CalibrationPara.rPitchCalib:=STRING_TO_REAL(sValue); END_IF;
				IF sVariableName = 'rplungelengthgrindfeedcalib' THEN ptrData_ProcessImageLoadData^.T_CalibrationPara.rPlungeLengthGrindFeedCalib:=STRING_TO_REAL(sValue); END_IF;
				IF sVariableName = 'rplungelengthtoolfeedcalib' THEN ptrData_ProcessImageLoadData^.T_CalibrationPara.rPlungeLengthToolFeedCalib:=STRING_TO_REAL(sValue); END_IF;
				IF sVariableName = 'rplungespeedgrindfeedcalib' THEN ptrData_ProcessImageLoadData^.T_CalibrationPara.rPlungeSpeedGrindFeedCalib:=STRING_TO_REAL(sValue); END_IF;
				IF sVariableName = 'rspeedtoolrotationcalib' THEN ptrData_ProcessImageLoadData^.T_CalibrationPara.rSpeedToolRotationCalib:=STRING_TO_REAL(sValue); END_IF;
				IF sVariableName = 'rstartpostoolfeedcalib' THEN ptrData_ProcessImageLoadData^.T_CalibrationPara.rStartPosToolFeedCalib:=STRING_TO_REAL(sValue); END_IF;
				IF sVariableName = 'rtoollengthcylinderpartcalib' THEN ptrData_ProcessImageLoadData^.T_CalibrationPara.rToolLengthCylinderPartCalib:=STRING_TO_REAL(sValue); END_IF;
				IF sVariableName = 'rdisplaceactivationcalib' THEN
					IF (STRING_TO_REAL(sValue) = 0) THEN
						ptrData_ProcessImageLoadData^.T_CalibrationPara.xDisplaceActivationCalib:=FALSE;
					ELSE
						ptrData_ProcessImageLoadData^.T_CalibrationPara.xDisplaceActivationCalib:=TRUE;
					END_IF;
				END_IF;
				IF sVariableName = 'rplungeactivationcalib' THEN
					IF (STRING_TO_REAL(sValue) = 0) THEN
						ptrData_ProcessImageLoadData^.T_CalibrationPara.xPlungeActivationCalib:=FALSE;
					ELSE
						ptrData_ProcessImageLoadData^.T_CalibrationPara.xPlungeActivationCalib:=TRUE;
					END_IF;
				END_IF;
				IF sVariableName = 'roffsetbeforetooldiagrindfeedprocess' THEN ptrData_ProcessImageLoadData^.T_ProcessPara.rOffsetBeforeToolDiaGrindFeedProcess:=STRING_TO_REAL(sValue); END_IF;
				IF sVariableName = 'rsecurityposgrindfeedprocess' THEN ptrData_ProcessImageLoadData^.T_ProcessPara.rSecurityPosGrindFeedProcess:=STRING_TO_REAL(sValue); END_IF;
				IF sVariableName = 'rspeedbackwardgrindfeed' THEN ptrData_ProcessImageLoadData^.T_ProcessPara.rSpeedBackwardGrindFeed:=STRING_TO_REAL(sValue); END_IF;
				IF sVariableName = 'rspeedforwardfastgrindfeed' THEN ptrData_ProcessImageLoadData^.T_ProcessPara.rSpeedForwardFastGrindFeed:=STRING_TO_REAL(sValue); END_IF;
				IF sVariableName = 'rspeedforwardslowgrindfeed' THEN ptrData_ProcessImageLoadData^.T_ProcessPara.rSpeedForwardSlowGrindFeed:=STRING_TO_REAL(sValue); END_IF;
				IF sVariableName = 'rspeedstartpostoolfeedprocess' THEN ptrData_ProcessImageLoadData^.T_ProcessPara.rSpeedStartPosToolFeedProcess:=STRING_TO_REAL(sValue); END_IF;
				IF sVariableName = 'rstartpostoolfeedauto' THEN ptrData_ProcessImageLoadData^.T_ProcessPara.rStartPosToolFeedAuto:=STRING_TO_REAL(sValue); END_IF;
				IF sVariableName = 'rtooldiameterprocess' THEN ptrData_ProcessImageLoadData^.T_ProcessPara.rToolDiameterProcess:=STRING_TO_REAL(sValue); END_IF;
				IF sVariableName = 'rtooltensionprocess' THEN ptrData_ProcessImageLoadData^.T_ProcessPara.rToolTensionProcess:=STRING_TO_REAL(sValue); END_IF;
		END_IF
	END_FOR
	(* confirm copy value *)
	xFctCopyDataFileToProfile:=TRUE;
END_FUNCTION

(* POU GENERAL/FB_CONTROLLAMP, ST *)
FUNCTION_BLOCK FB_CONTROLLAMP
VAR_INPUT
	xStartUpCompleted:BOOL;		(* State of the machine, if the booting of the machine is active *)
	iStateMessage:INT;			(* State of the message-->with the number 401, an error occur *)
	bActiveStation:BYTE;			(* 0=Normalbetrieb, 1,2,3,4=Sonderbetrieb *)
END_VAR
VAR_IN_OUT
	T_Station:ST_STATION;		(* Data structure of the station level *)
	T_Process : ST_PROCESS;	(* Data structure of the process level *)
	TCtrlePanel:ST_CTRLEPANEL;	(* Data structure of the ControlPanel *)
END_VAR
VAR_OUTPUT
	xLampGreen:BOOL;			(* Output signal for the green lamp *)
	xLampRed:BOOL;				(* Output signal for the red lamp *)
	xLampOrange:BOOL;			(* Output signal for the orange lamp *)
END_VAR
VAR
(* Timer *)
	TimerON:TON;
	TimerOFF:TOF;
	tTimerCadence:TIME;
	xTimerSignal:BOOL;
(* variable *)
	xFirstExecution:BOOL;
	xRedOffGreenOff:BOOL;
	xRedOnGreenOff:BOOL;
	xRedBlinkedGreenOff:BOOL;
	xRedOffGreenOn:BOOL;
	xRedOffGreenBlinked:BOOL;
	xRedOnGreenOn:BOOL;
	xRedAndGreenBlinked: BOOL;
	xPanelLedBlinked: BOOL;
(* Tmp *)
	xTmp:BOOL;
END_VAR
(****************************************************************************************************************************************************)
(***********                             This Functionblock set the ControlLamp for the different state of the machine                                ************)
(****************************************************************************************************************************************************)
(* First execution *)
	IF NOT xFirstExecution THEN
		(* Init. variable *)
		tTimerCadence:=T#0.5s;
		xTimerSignal:=FALSE;
		(* Timer *)
		TimerON(IN:=FALSE);
		TimerOFF(IN:=TRUE);
		(* Confirm execution *)
		xFirstExecution:=TRUE;
	END_IF

(* Each cycle, init. lamp state *)
	xLampGreen:=FALSE;
	xLampRed:=FALSE;
	xLampOrange:=FALSE;
	TCtrlePanel.udiLED:=16#0;

(* Each cycle, init. lamp state function *)
	xTmp:=FALSE;
	xRedOffGreenOff:=FALSE;
	xRedOnGreenOff:=FALSE;
	xRedBlinkedGreenOff:=FALSE;
	xRedOffGreenOn:=FALSE;
	xRedOffGreenBlinked:=FALSE;
	xRedOnGreenOn:=FALSE;
	xRedAndGreenBlinked:=FALSE;
	xPanelLedBlinked:=FALSE;

(* Error *)
	IF NOT(xStartUpCompleted) THEN
		(* While starting up of the machine *)
		 xRedOnGreenOn:=TRUE;
	ELSE
		IF (iStateMessage = 401) THEN
			(* Error state *)
			xRedBlinkedGreenOff:=TRUE;
			xPanelLedBlinked:=TRUE;
		ELSIF NOT(T_Process.xEnd) AND ((T_Process.iFunctNr = 10) OR (T_Process.iFunctNr = 20) OR (T_Process.iFunctNr = 30)) THEN
			(* Normalbetrieb with active process *)
			xRedOffGreenOn:=TRUE;
		ELSIF T_Process.xEnd AND (bActiveStation = 0) THEN
			(* Normalbetrieb and no active process *)
			xRedOffGreenBlinked:=TRUE;
		ELSIF (bActiveStation <> 0) THEN
			(* Einrichtbetrieb *)
			xRedAndGreenBlinked:=TRUE;
		ELSE
			(* Dieser Zustand sollte niemals eintreten dürfen *)
			xRedOffGreenOff:=TRUE;
		END_IF;
	END_IF;

(* Blink *)
	TimerON(IN:=TRUE,PT:=tTimerCadence);
	IF TimerON.Q THEN
		TimerOFF(IN:=FALSE,PT:=tTimerCadence);
		IF NOT TimerOFF.Q THEN TimerON(IN:=FALSE); TimerOFF(IN:=TRUE); END_IF
	END_IF

(* Red off and green off *)
	IF xRedOffGreenOff THEN
		xLampGreen:=FALSE;
		xLampRed:=FALSE;
	END_IF

(* Red on and green off *)
	IF xRedOnGreenOff THEN
		xLampGreen:=FALSE;
		xLampRed:=TRUE;
	END_IF

(* Red blinked green off *)
	IF xRedBlinkedGreenOff THEN
		xLampGreen:=FALSE;
		xLampRed:=TimerON.Q;
		tTimerCadence:=T#0.5s;
	END_IF

(* Red off green on *)
	IF xRedOffGreenOn THEN
		xLampGreen:=TRUE;
		xLampRed:=FALSE;
	END_IF

(* Red off green blinked *)
	IF xRedOffGreenBlinked THEN
		xLampGreen:=TimerON.Q;
		tTimerCadence:=T#0.5s;
		xLampRed:=FALSE;
	END_IF

(* Red on green on *)
	IF xRedOnGreenOn THEN
		xLampGreen:=TRUE;
		xLampRed:=TRUE;
	END_IF

(* Red and green blinked *)
	IF xRedAndGreenBlinked THEN
		xLampGreen:=TimerON.Q;
		xLampRed:=xLampGreen;
		tTimerCadence:=T#0.5s;
	END_IF

(* Panel led blinked *)
	IF xPanelLedBlinked THEN
		IF TimerON.Q THEN TCtrlePanel.udiLED:=16#3FF; ELSE TCtrlePanel.udiLED:=16#0; END_IF
	END_IF
END_FUNCTION_BLOCK

(* POU PRG_HARDWARE_LAYER2/PRG_HW_STATION, FBD *)
PROGRAM PRG_HW_STATION
VAR
	FBHWStation: FBHW_STATION;

(* Ecostep PDO Parameter *)
	TToolLeftRxPdoPara AT %Q*:ST_RX_PDO_PARA;
	TToolLeftTxPdoPara AT %I*:ST_TX_PDO_PARA;
	TToolCenterRxPdoPara AT %Q*:ST_RX_PDO_PARA;
	TToolCenterTxPdoPara AT %I*:ST_TX_PDO_PARA;
	TToolRightRxPdoPara AT %Q*:ST_RX_PDO_PARA;
	TToolRightTxPdoPara AT %I*:ST_TX_PDO_PARA;
	TToolFeederRxPdoPara AT %Q*:ST_RX_PDO_PARA;
	TToolFeederTxPdoPara AT %I*:ST_TX_PDO_PARA;
	TGrindFeederRxPdoPara AT %Q*:ST_RX_PDO_PARA;
	TGrindFeederTxPdoPara AT %I*:ST_TX_PDO_PARA;

(* Beckhoff Axis structure *)
	stToolLeftRefOut AT %Q* :PLCTONC_AXLESTRUCT;
	stToolLeftRefIn AT %I* :NCTOPLC_AXLESTRUCT;
	stToolCenterRefOut AT %Q* :PLCTONC_AXLESTRUCT;
	stToolCenterRefIn AT %I* :NCTOPLC_AXLESTRUCT;
	stToolRightRefOut AT %Q* :PLCTONC_AXLESTRUCT;
	stToolRightRefIn AT %I* :NCTOPLC_AXLESTRUCT;
	stToolFeederRefOut AT %Q* :PLCTONC_AXLESTRUCT;
	stToolFeederRefIn AT %I* :NCTOPLC_AXLESTRUCT;
	stGrindFeederRefOut AT %Q* :PLCTONC_AXLESTRUCT;
	stGrindFeederRefIn AT %I* :NCTOPLC_AXLESTRUCT;

	auiActualAxisTorqueBeckhoff AT %I*:ARRAY [1..5] OF UINT;
	axInputAxisBeckhoff AT %I*: ARRAY[1..5,1..8] OF BOOL;
END_VAR
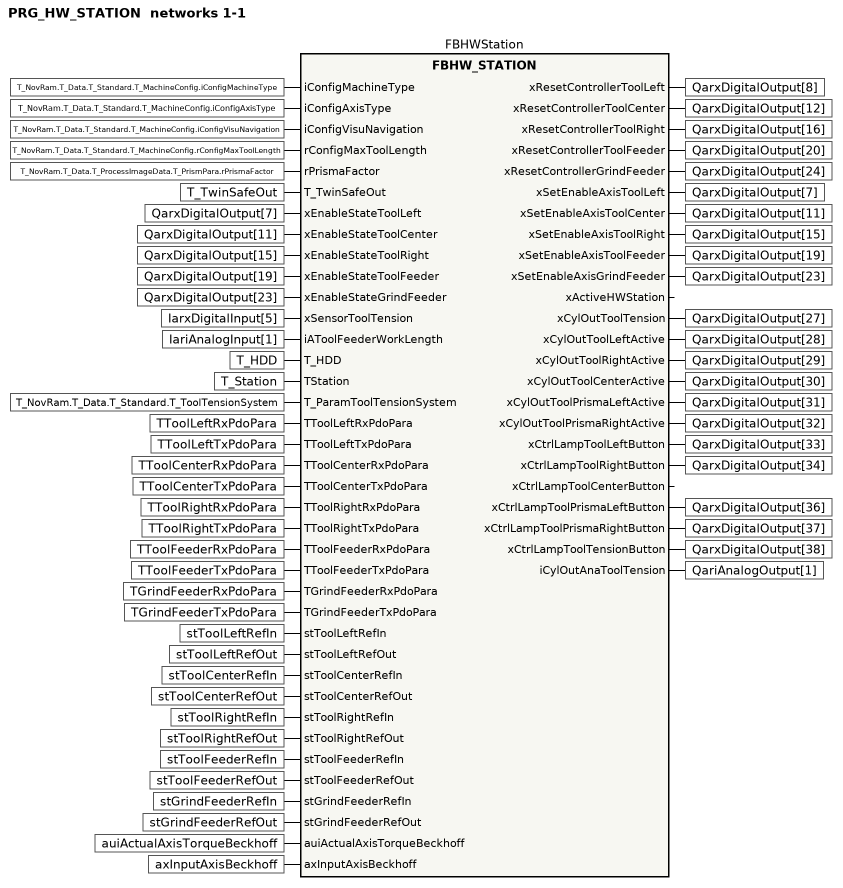
_FBD_ (* Function Block Diagram *)
NETWORK 1 (* HARDWARE LEVEL-->LAYER 2 *)
	FBHWStation:FBHW_STATION(iConfigMachineType: T_NovRam.T_Data.T_Standard.T_MachineConfig.iConfigMachineType, iConfigAxisType: T_NovRam.T_Data.T_Standard.T_MachineConfig.iConfigAxisType, iConfigVisuNavigation: T_NovRam.T_Data.T_Standard.T_MachineConfig.iConfigVisuNavigation, rConfigMaxToolLength: T_NovRam.T_Data.T_Standard.T_MachineConfig.rConfigMaxToolLength, rPrismaFactor: T_NovRam.T_Data.T_ProcessImageData.T_PrismPara.rPrismaFactor, T_TwinSafeOut: T_TwinSafeOut, xEnableStateToolLeft: QarxDigitalOutput[7], xEnableStateToolCenter: QarxDigitalOutput[11], xEnableStateToolRight: QarxDigitalOutput[15], xEnableStateToolFeeder: QarxDigitalOutput[19], xEnableStateGrindFeeder: QarxDigitalOutput[23], xSensorToolTension: IarxDigitalInput[5], iAToolFeederWorkLength: IariAnalogInput[1], T_HDD: T_HDD, TStation: T_Station, T_ParamToolTensionSystem: T_NovRam.T_Data.T_Standard.T_ToolTensionSystem, TToolLeftRxPdoPara: TToolLeftRxPdoPara, TToolLeftTxPdoPara: TToolLeftTxPdoPara, TToolCenterRxPdoPara: TToolCenterRxPdoPara, TToolCenterTxPdoPara: TToolCenterTxPdoPara, TToolRightRxPdoPara: TToolRightRxPdoPara, TToolRightTxPdoPara: TToolRightTxPdoPara, TToolFeederRxPdoPara: TToolFeederRxPdoPara, TToolFeederTxPdoPara: TToolFeederTxPdoPara, TGrindFeederRxPdoPara: TGrindFeederRxPdoPara, TGrindFeederTxPdoPara: TGrindFeederTxPdoPara, stToolLeftRefIn: stToolLeftRefIn, stToolLeftRefOut: stToolLeftRefOut, stToolCenterRefIn: stToolCenterRefIn, stToolCenterRefOut: stToolCenterRefOut, stToolRightRefIn: stToolRightRefIn, stToolRightRefOut: stToolRightRefOut, stToolFeederRefIn: stToolFeederRefIn, stToolFeederRefOut: stToolFeederRefOut, stGrindFeederRefIn: stGrindFeederRefIn, stGrindFeederRefOut: stGrindFeederRefOut, auiActualAxisTorqueBeckhoff: auiActualAxisTorqueBeckhoff, axInputAxisBeckhoff: axInputAxisBeckhoff, xResetControllerToolCenter => QarxDigitalOutput[12], xResetControllerToolRight => QarxDigitalOutput[16], xResetControllerToolFeeder => QarxDigitalOutput[20], xResetControllerGrindFeeder => QarxDigitalOutput[24], xSetEnableAxisToolLeft => QarxDigitalOutput[7], xSetEnableAxisToolCenter => QarxDigitalOutput[11], xSetEnableAxisToolRight => QarxDigitalOutput[15], xSetEnableAxisToolFeeder => QarxDigitalOutput[19], xSetEnableAxisGrindFeeder => QarxDigitalOutput[23], xCylOutToolTension => QarxDigitalOutput[27], xCylOutToolLeftActive => QarxDigitalOutput[28], xCylOutToolRightActive => QarxDigitalOutput[29], xCylOutToolCenterActive => QarxDigitalOutput[30], xCylOutToolPrismaLeftActive => QarxDigitalOutput[31], xCylOutToolPrismaRightActive => QarxDigitalOutput[32], xCtrlLampToolLeftButton => QarxDigitalOutput[33], xCtrlLampToolRightButton => QarxDigitalOutput[34], xCtrlLampToolPrismaLeftButton => QarxDigitalOutput[36], xCtrlLampToolPrismaRightButton => QarxDigitalOutput[37], xCtrlLampToolTensionButton => QarxDigitalOutput[38], iCylOutAnaToolTension => QariAnalogOutput[1]) => QarxDigitalOutput[8]
_END_FBD_
(* the same logic as Structured Text *)
(* Network 1: HARDWARE LEVEL-->LAYER 2 *)
FBHWStation(iConfigMachineType := T_NovRam.T_Data.T_Standard.T_MachineConfig.iConfigMachineType, iConfigAxisType := T_NovRam.T_Data.T_Standard.T_MachineConfig.iConfigAxisType, iConfigVisuNavigation := T_NovRam.T_Data.T_Standard.T_MachineConfig.iConfigVisuNavigation, rConfigMaxToolLength := T_NovRam.T_Data.T_Standard.T_MachineConfig.rConfigMaxToolLength, rPrismaFactor := T_NovRam.T_Data.T_ProcessImageData.T_PrismPara.rPrismaFactor, T_TwinSafeOut := T_TwinSafeOut, xEnableStateToolLeft := QarxDigitalOutput[7], xEnableStateToolCenter := QarxDigitalOutput[11], xEnableStateToolRight := QarxDigitalOutput[15], xEnableStateToolFeeder := QarxDigitalOutput[19], xEnableStateGrindFeeder := QarxDigitalOutput[23], xSensorToolTension := IarxDigitalInput[5], iAToolFeederWorkLength := IariAnalogInput[1], T_HDD := T_HDD, TStation := T_Station, T_ParamToolTensionSystem := T_NovRam.T_Data.T_Standard.T_ToolTensionSystem, TToolLeftRxPdoPara := TToolLeftRxPdoPara, TToolLeftTxPdoPara := TToolLeftTxPdoPara, TToolCenterRxPdoPara := TToolCenterRxPdoPara, TToolCenterTxPdoPara := TToolCenterTxPdoPara, TToolRightRxPdoPara := TToolRightRxPdoPara, TToolRightTxPdoPara := TToolRightTxPdoPara, TToolFeederRxPdoPara := TToolFeederRxPdoPara, TToolFeederTxPdoPara := TToolFeederTxPdoPara, TGrindFeederRxPdoPara := TGrindFeederRxPdoPara, TGrindFeederTxPdoPara := TGrindFeederTxPdoPara, stToolLeftRefIn := stToolLeftRefIn, stToolLeftRefOut := stToolLeftRefOut, stToolCenterRefIn := stToolCenterRefIn, stToolCenterRefOut := stToolCenterRefOut, stToolRightRefIn := stToolRightRefIn, stToolRightRefOut := stToolRightRefOut, stToolFeederRefIn := stToolFeederRefIn, stToolFeederRefOut := stToolFeederRefOut, stGrindFeederRefIn := stGrindFeederRefIn, stGrindFeederRefOut := stGrindFeederRefOut, auiActualAxisTorqueBeckhoff := auiActualAxisTorqueBeckhoff, axInputAxisBeckhoff := axInputAxisBeckhoff);
QarxDigitalOutput[12] := FBHWStation.xResetControllerToolCenter;
QarxDigitalOutput[16] := FBHWStation.xResetControllerToolRight;
QarxDigitalOutput[20] := FBHWStation.xResetControllerToolFeeder;
QarxDigitalOutput[24] := FBHWStation.xResetControllerGrindFeeder;
QarxDigitalOutput[7] := FBHWStation.xSetEnableAxisToolLeft;
QarxDigitalOutput[11] := FBHWStation.xSetEnableAxisToolCenter;
QarxDigitalOutput[15] := FBHWStation.xSetEnableAxisToolRight;
QarxDigitalOutput[19] := FBHWStation.xSetEnableAxisToolFeeder;
QarxDigitalOutput[23] := FBHWStation.xSetEnableAxisGrindFeeder;
QarxDigitalOutput[27] := FBHWStation.xCylOutToolTension;
QarxDigitalOutput[28] := FBHWStation.xCylOutToolLeftActive;
QarxDigitalOutput[29] := FBHWStation.xCylOutToolRightActive;
QarxDigitalOutput[30] := FBHWStation.xCylOutToolCenterActive;
QarxDigitalOutput[31] := FBHWStation.xCylOutToolPrismaLeftActive;
QarxDigitalOutput[32] := FBHWStation.xCylOutToolPrismaRightActive;
QarxDigitalOutput[33] := FBHWStation.xCtrlLampToolLeftButton;
QarxDigitalOutput[34] := FBHWStation.xCtrlLampToolRightButton;
QarxDigitalOutput[36] := FBHWStation.xCtrlLampToolPrismaLeftButton;
QarxDigitalOutput[37] := FBHWStation.xCtrlLampToolPrismaRightButton;
QarxDigitalOutput[38] := FBHWStation.xCtrlLampToolTensionButton;
QariAnalogOutput[1] := FBHWStation.iCylOutAnaToolTension;
QarxDigitalOutput[8] := FBHWStation.xResetControllerToolLeft;
END_PROGRAM

(* POU PRG_HARDWARE_LAYER2/FBHWSTATIONEN/FBHW_STATION, ST *)
FUNCTION_BLOCK FBHW_STATION
VAR_INPUT
	iConfigMachineType:INT;				(* Machine config parameter, 1=MicroWire, 2=MicroRod *)
	iConfigAxisType:INT;					(* Machine config parameter, 1=EcoStep Axis, 2=Beckhoff Axis *)
	iConfigVisuNavigation:INT;				(* Machine config parameter, 1=left and right special button are active, 2=left and right touchbutton are active  *)
	rConfigMaxToolLength:REAL;			(* Machine config parameter, input of the maximal to worked tool length *)
	rPrismaFactor:REAL;					(* correction value of the GrindFeeder axis, this is depend of the settled prisma *)
	T_TwinSafeOut:ST_TWINSAFE_OUT;	(* Output of the TwinSafe components *)
	xEnableStateToolLeft:BOOL;			(* Enable state of the ToolLeft axis *)
	xEnableStateToolCenter:BOOL;			(* Enable state of the ToolCenter axis *)
	xEnableStateToolRight:BOOL;			(* Enable state of the ToolRight axis *)
	xEnableStateToolFeeder:BOOL;			(* Enable state of the ToolFeeder axis *)
	xEnableStateGrindFeeder:BOOL;		(* Enable state of the GrindFeeder axis *)
	xSensorToolTension:BOOL;			(* Signal of the sensor for the ToolTension-->this is only for the MicroRod *)
	iAToolFeederWorkLength:INT;			(* Signal for measuring the max work length of the ToolFeeder *)
END_VAR
VAR_IN_OUT
	T_HDD : ST_HDD;					(* Data structure of the file management *)
	TStation:ST_STATION;				(* Data structure of the Stationlevel *)
	T_ParamToolTensionSystem:ST_EXCHG_PARAM_TOOLTENSIONSYSTEM;	(* NovRam parameter of the ToolTension *)
	(* Ecostep PDO Parameter *)
	TToolLeftRxPdoPara:ST_RX_PDO_PARA;
	TToolLeftTxPdoPara:ST_TX_PDO_PARA;
	TToolCenterRxPdoPara:ST_RX_PDO_PARA;
	TToolCenterTxPdoPara:ST_TX_PDO_PARA;
	TToolRightRxPdoPara:ST_RX_PDO_PARA;
	TToolRightTxPdoPara:ST_TX_PDO_PARA;
	TToolFeederRxPdoPara:ST_RX_PDO_PARA;
	TToolFeederTxPdoPara:ST_TX_PDO_PARA;
	TGrindFeederRxPdoPara:ST_RX_PDO_PARA;
	TGrindFeederTxPdoPara:ST_TX_PDO_PARA;
	(* Beckhoff Axis structure *)
	stToolLeftRefIn :NCTOPLC_AXLESTRUCT;
	stToolLeftRefOut :PLCTONC_AXLESTRUCT;
	stToolCenterRefIn :NCTOPLC_AXLESTRUCT;
	stToolCenterRefOut :PLCTONC_AXLESTRUCT;
	stToolRightRefIn :NCTOPLC_AXLESTRUCT;
	stToolRightRefOut :PLCTONC_AXLESTRUCT;
	stToolFeederRefIn :NCTOPLC_AXLESTRUCT;
	stToolFeederRefOut :PLCTONC_AXLESTRUCT;
	stGrindFeederRefIn :NCTOPLC_AXLESTRUCT;
	stGrindFeederRefOut :PLCTONC_AXLESTRUCT;
	auiActualAxisTorqueBeckhoff:ARRAY [1..5] OF UINT;
	axInputAxisBeckhoff : ARRAY[1..5,1..8] OF BOOL;
END_VAR
VAR_OUTPUT
	xResetControllerToolLeft:BOOL;			(* Reset output for the ToolLeft axis *)
	xResetControllerToolCenter:BOOL;		(* Reset output for the ToolCenter axis *)
	xResetControllerToolRight:BOOL;		(* Reset output for the ToolRight axis *)
	xResetControllerToolFeeder:BOOL;		(* Reset output for the ToolFeeder axis *)
	xResetControllerGrindFeeder:BOOL;		(* Reset output for the GrindFeeder axis *)
	xSetEnableAxisToolLeft:BOOL;			(* Enable output for the ToolLeft axis *)
	xSetEnableAxisToolCenter:BOOL;		(* Enable output for the ToolCenter axis *)
	xSetEnableAxisToolRight:BOOL;			(* Enable output for the ToolRight axis *)
	xSetEnableAxisToolFeeder:BOOL;		(* Enable output for the ToolFeeder axis *)
	xSetEnableAxisGrindFeeder:BOOL;		(* Enable output for the GrindFeeder axis *)
	xActiveHWStation : BOOL;				(* state of the activation of the station hardware *)
	xCylOutToolTension : BOOL;			(* ventil for the Cylinder ToolTension *)
(*22.12.2009: KFS {    *)
	xCylOutToolLeftActive : BOOL;			(* ventil for the Cylinder ToolLeft *)
	xCylOutToolRightActive: BOOL;			(* ventil for the Cylinder ToolRight *)
	xCylOutToolCenterActive : BOOL;		(* ventil for the Cylinder ToolCenter *)
	xCylOutToolPrismaLeftActive : BOOL;		(* ventil for the Cylinder ToolPrismaLeft *)
	xCylOutToolPrismaRightActive : BOOL;	(* ventil for the Cylinder ToolPrismaRight *)
	xCtrlLampToolLeftButton : BOOL;			(* control lamp button for the Cylinder ToolLeft *)
	xCtrlLampToolRightButton : BOOL;		(* control lamp button for the Cylinder ToolRight*)
	xCtrlLampToolCenterButton : BOOL;		(* control lamp button for the Cylinder ToolCenter *)
	xCtrlLampToolPrismaLeftButton : BOOL;	(* control lamp button for the Cylinder ToolPrismaLeft *)
	xCtrlLampToolPrismaRightButton : BOOL;	(* control lamp button for the Cylinder ToolPrismaRight *)
	xCtrlLampToolTensionButton : BOOL;		(* control lamp button for the Cylinder ToolTension *)
(*22.12.2009: KFS }    *)
	iCylOutAnaToolTension : INT;			(* servoventil for the Cylinder ToolTension *)
END_VAR
VAR
(* Ecostep Driver *)
	FBAxisToolLeftEcostep: FBHW_AXIS_SINGLE_ECOSTEP;
	FBAxisToolCenterEcostep: FBHW_AXIS_SINGLE_ECOSTEP;
	FBAxisToolRightEcostep: FBHW_AXIS_SINGLE_ECOSTEP;
	FBAxisToolFeederEcostep: FBHW_AXIS_SINGLE_ECOSTEP;
	FBAxisGrindFeederEcostep: FBHW_AXIS_SINGLE_ECOSTEP;
	FBLivevalueAxisToolLeftEcostep: FBHW_AXIS_LIVEVALUES_ECOSTEP;
	FBLivevalueAxisToolCenterEcostep: FBHW_AXIS_LIVEVALUES_ECOSTEP;
	FBLivevalueAxisToolRightEcostep: FBHW_AXIS_LIVEVALUES_ECOSTEP;
	FBLivevalueAxisToolFeederEcostep: FBHW_AXIS_LIVEVALUES_ECOSTEP;
	FBLivevalueAxisGrindFeederEcostep: FBHW_AXIS_LIVEVALUES_ECOSTEP;

